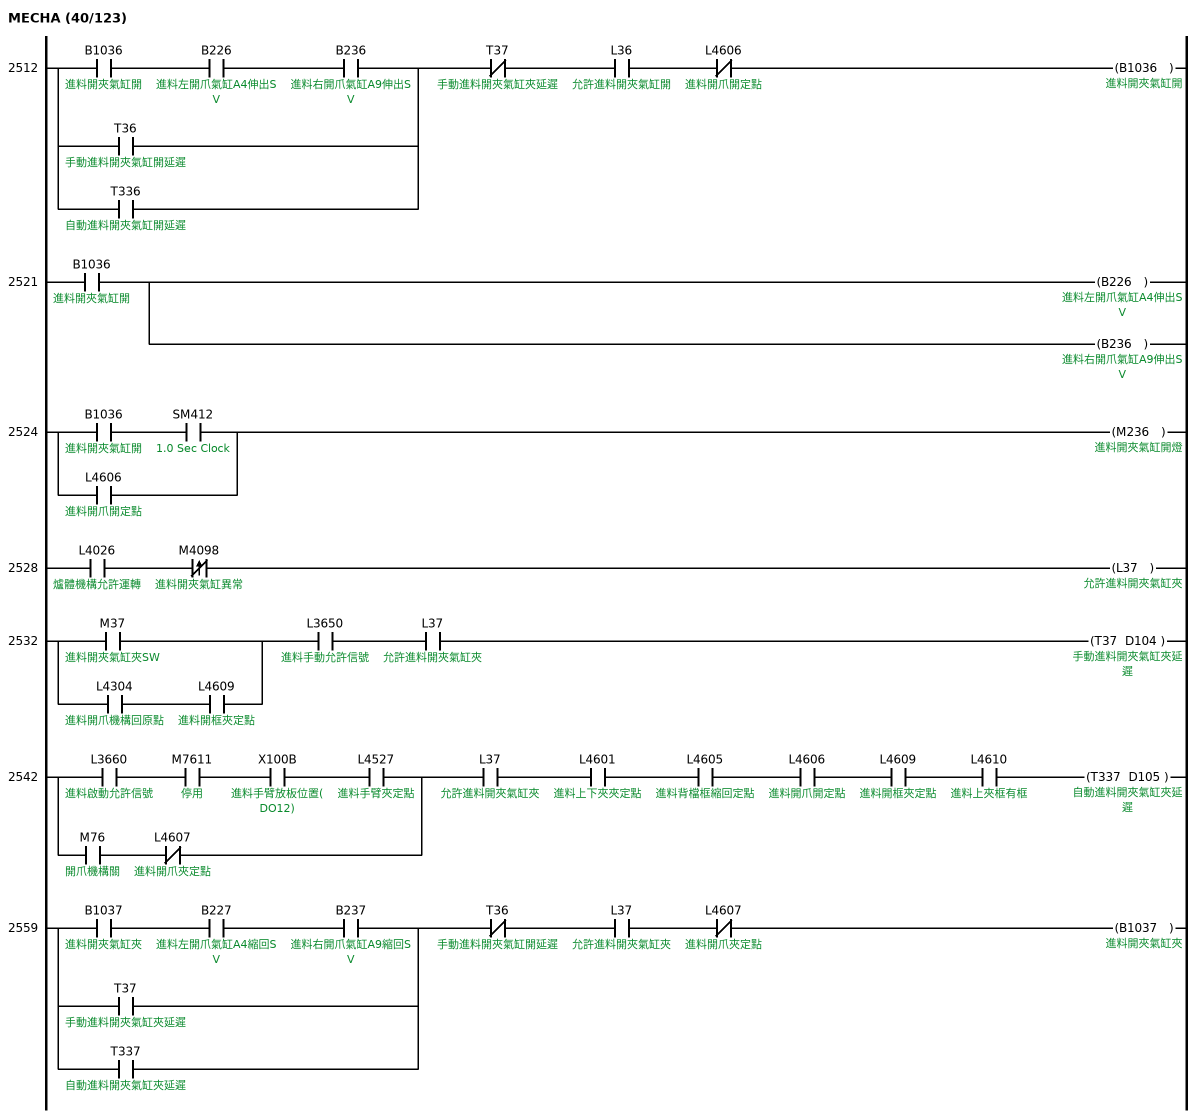
[picture p336: ladder of MECHA, rungs at steps 2512 to 2559]
2512  LD      B1036  ; 進料開夾氣缸開
      AND     B226  ; 進料左開爪氣缸A4伸出SV
      AND     B236  ; 進料右開爪氣缸A9伸出SV
      OR      T36  ; 手動進料開夾氣缸開延遲
      OR      T336  ; 自動進料開夾氣缸開延遲
      ANI     T37  ; 手動進料開夾氣缸夾延遲
      AND     L36  ; 允許進料開夾氣缸開
      ANI     L4606  ; 進料開爪開定點
      OUT     B1036  ; 進料開夾氣缸開
2521  LD      B1036  ; 進料開夾氣缸開
      OUT     B226  ; 進料左開爪氣缸A4伸出SV
      OUT     B236  ; 進料右開爪氣缸A9伸出SV
2524  LD      B1036  ; 進料開夾氣缸開
      AND     SM412  ; 1.0 Sec Clock
      OR      L4606  ; 進料開爪開定點
      OUT     M236  ; 進料開夾氣缸開燈
2528  LD      L4026  ; 爐體機構允許運轉
      ANDPI   M4098  ; 進料開夾氣缸異常
      OUT     L37  ; 允許進料開夾氣缸夾
2532  LD      M37  ; 進料開夾氣缸夾SW
      LD      L4304  ; 進料開爪機構回原點
      AND     L4609  ; 進料開框夾定點
      ORB
      AND     L3650  ; 進料手動允許信號
      AND     L37  ; 允許進料開夾氣缸夾
      OUT     T37 D104  ; 手動進料開夾氣缸夾延遲
2542  LD      L3660  ; 進料啟動允許信號
      AND     M7611  ; 停用
      AND     X100B  ; 進料手臂放板位置(DO12)
      AND     L4527  ; 進料手臂夾定點
      LD      M76  ; 開爪機構關
      ANI     L4607  ; 進料開爪夾定點
      ORB
      AND     L37  ; 允許進料開夾氣缸夾
      AND     L4601  ; 進料上下夾夾定點
      AND     L4605  ; 進料背檔框縮回定點
      AND     L4606  ; 進料開爪開定點
      AND     L4609  ; 進料開框夾定點
      AND     L4610  ; 進料上夾框有框
      OUT     T337 D105  ; 自動進料開夾氣缸夾延遲
2559  LD      B1037  ; 進料開夾氣缸夾
      AND     B227  ; 進料左開爪氣缸A4縮回SV
      AND     B237  ; 進料右開爪氣缸A9縮回SV
      OR      T37  ; 手動進料開夾氣缸夾延遲
      OR      T337  ; 自動進料開夾氣缸夾延遲
      ANI     T36  ; 手動進料開夾氣缸開延遲
      AND     L37  ; 允許進料開夾氣缸夾
      ANI     L4607  ; 進料開爪夾定點
      OUT     B1037  ; 進料開夾氣缸夾
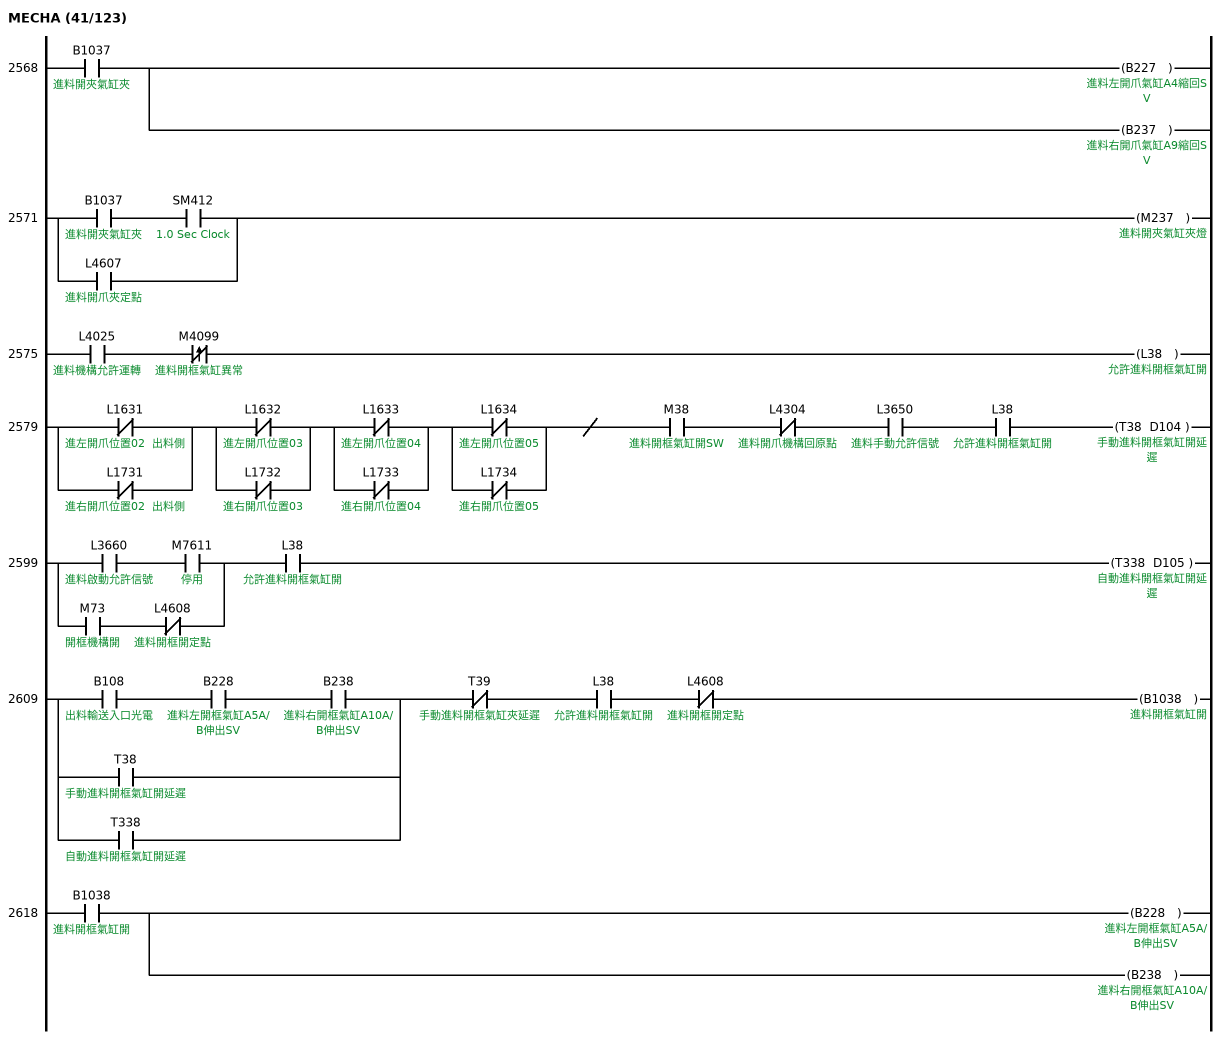
2568  LD      B1037  ; 進料開夾氣缸夾
      OUT     B227  ; 進料左開爪氣缸A4縮回SV
      OUT     B237  ; 進料右開爪氣缸A9縮回SV
2571  LD      B1037  ; 進料開夾氣缸夾
      AND     SM412  ; 1.0 Sec Clock
      OR      L4607  ; 進料開爪夾定點
      OUT     M237  ; 進料開夾氣缸夾燈
2575  LD      L4025  ; 進料機構允許運轉
      ANDPI   M4099  ; 進料開框氣缸異常
      OUT     L38  ; 允許進料開框氣缸開
2579  LDI     L1631  ; 進左開爪位置02  出料側
      ORI     L1731  ; 進右開爪位置02  出料側
      LDI     L1632  ; 進左開爪位置03
      ORI     L1732  ; 進右開爪位置03
      ANB
      LDI     L1633  ; 進左開爪位置04
      ORI     L1733  ; 進右開爪位置04
      ANB
      LDI     L1634  ; 進左開爪位置05
      ORI     L1734  ; 進右開爪位置05
      ANB
      INV
      AND     M38  ; 進料開框氣缸開SW
      ANI     L4304  ; 進料開爪機構回原點
      AND     L3650  ; 進料手動允許信號
      AND     L38  ; 允許進料開框氣缸開
      OUT     T38 D104  ; 手動進料開框氣缸開延遲
2599  LD      L3660  ; 進料啟動允許信號
      AND     M7611  ; 停用
      LD      M73  ; 開框機構開
      ANI     L4608  ; 進料開框開定點
      ORB
      AND     L38  ; 允許進料開框氣缸開
      OUT     T338 D105  ; 自動進料開框氣缸開延遲
2609  LD      B108  ; 出料輸送入口光電
      AND     B228  ; 進料左開框氣缸A5A/B伸出SV
      AND     B238  ; 進料右開框氣缸A10A/B伸出SV
      OR      T38  ; 手動進料開框氣缸開延遲
      OR      T338  ; 自動進料開框氣缸開延遲
      ANI     T39  ; 手動進料開框氣缸夾延遲
      AND     L38  ; 允許進料開框氣缸開
      ANI     L4608  ; 進料開框開定點
      OUT     B1038  ; 進料開框氣缸開
2618  LD      B1038  ; 進料開框氣缸開
      OUT     B228  ; 進料左開框氣缸A5A/B伸出SV
      OUT     B238  ; 進料右開框氣缸A10A/B伸出SV
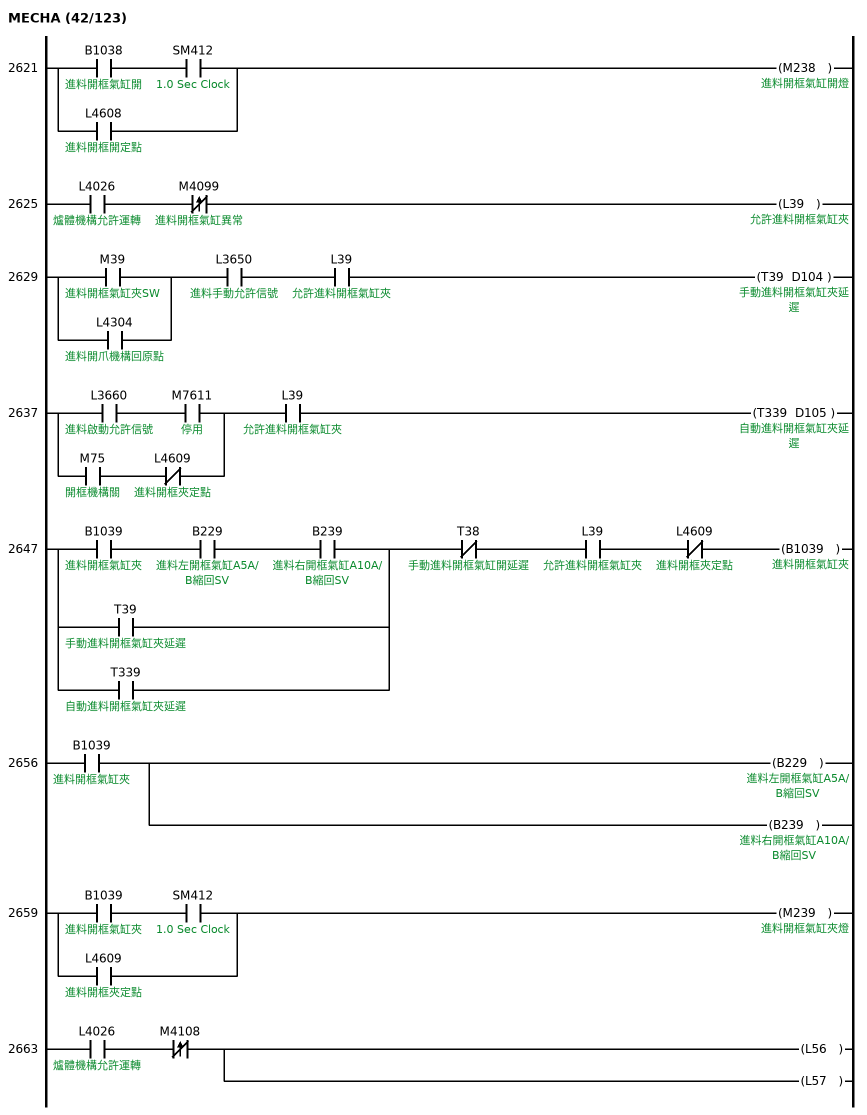
2621  LD      B1038  ; 進料開框氣缸開
      AND     SM412  ; 1.0 Sec Clock
      OR      L4608  ; 進料開框開定點
      OUT     M238  ; 進料開框氣缸開燈
2625  LD      L4026  ; 爐體機構允許運轉
      ANDPI   M4099  ; 進料開框氣缸異常
      OUT     L39  ; 允許進料開框氣缸夾
2629  LD      M39  ; 進料開框氣缸夾SW
      OR      L4304  ; 進料開爪機構回原點
      AND     L3650  ; 進料手動允許信號
      AND     L39  ; 允許進料開框氣缸夾
      OUT     T39 D104  ; 手動進料開框氣缸夾延遲
2637  LD      L3660  ; 進料啟動允許信號
      AND     M7611  ; 停用
      LD      M75  ; 開框機構關
      ANI     L4609  ; 進料開框夾定點
      ORB
      AND     L39  ; 允許進料開框氣缸夾
      OUT     T339 D105  ; 自動進料開框氣缸夾延遲
2647  LD      B1039  ; 進料開框氣缸夾
      AND     B229  ; 進料左開框氣缸A5A/B縮回SV
      AND     B239  ; 進料右開框氣缸A10A/B縮回SV
      OR      T39  ; 手動進料開框氣缸夾延遲
      OR      T339  ; 自動進料開框氣缸夾延遲
      ANI     T38  ; 手動進料開框氣缸開延遲
      AND     L39  ; 允許進料開框氣缸夾
      ANI     L4609  ; 進料開框夾定點
      OUT     B1039  ; 進料開框氣缸夾
2656  LD      B1039  ; 進料開框氣缸夾
      OUT     B229  ; 進料左開框氣缸A5A/B縮回SV
      OUT     B239  ; 進料右開框氣缸A10A/B縮回SV
2659  LD      B1039  ; 進料開框氣缸夾
      AND     SM412  ; 1.0 Sec Clock
      OR      L4609  ; 進料開框夾定點
      OUT     M239  ; 進料開框氣缸夾燈
2663  LD      L4026  ; 爐體機構允許運轉
      ANDPI   M4108
      OUT     L56
      OUT     L57
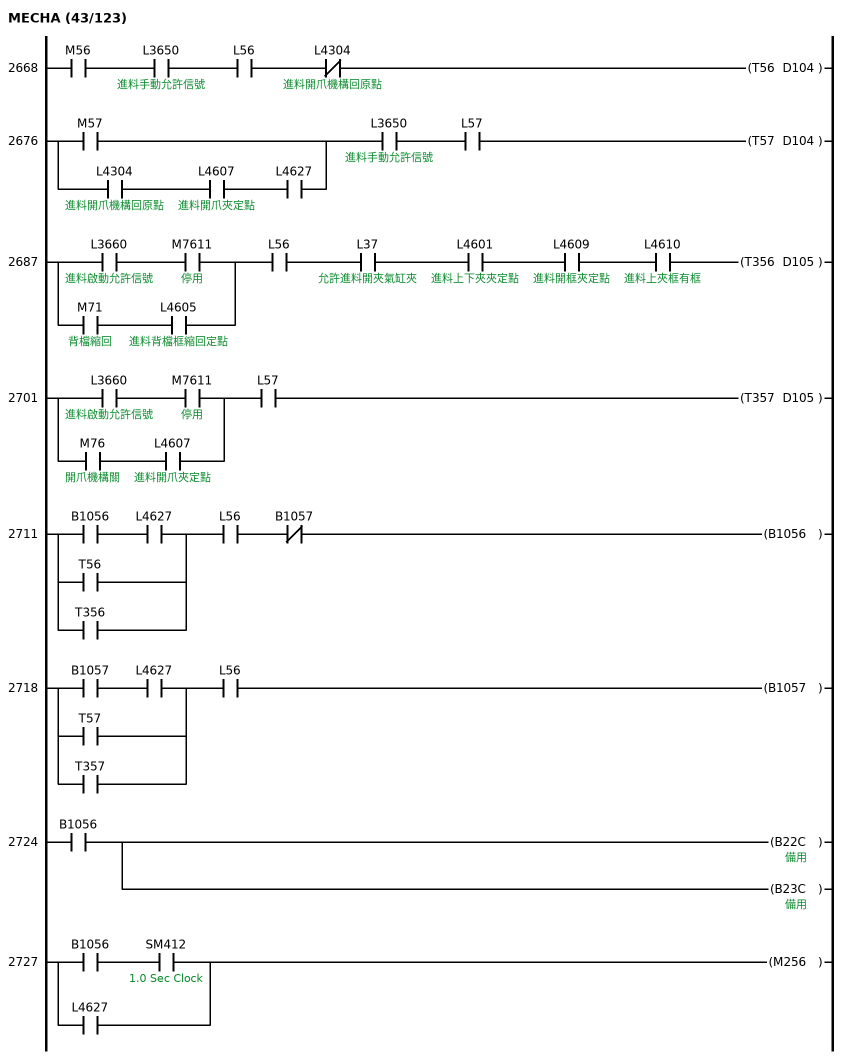
2668  LD      M56
      AND     L3650  ; 進料手動允許信號
      AND     L56
      ANI     L4304  ; 進料開爪機構回原點
      OUT     T56 D104
2676  LD      M57
      LD      L4304  ; 進料開爪機構回原點
      AND     L4607  ; 進料開爪夾定點
      AND     L4627
      ORB
      AND     L3650  ; 進料手動允許信號
      AND     L57
      OUT     T57 D104
2687  LD      L3660  ; 進料啟動允許信號
      AND     M7611  ; 停用
      LD      M71  ; 背檔縮回
      AND     L4605  ; 進料背檔框縮回定點
      ORB
      AND     L56
      AND     L37  ; 允許進料開夾氣缸夾
      AND     L4601  ; 進料上下夾夾定點
      AND     L4609  ; 進料開框夾定點
      AND     L4610  ; 進料上夾框有框
      OUT     T356 D105
2701  LD      L3660  ; 進料啟動允許信號
      AND     M7611  ; 停用
      LD      M76  ; 開爪機構關
      AND     L4607  ; 進料開爪夾定點
      ORB
      AND     L57
      OUT     T357 D105
2711  LD      B1056
      AND     L4627
      OR      T56
      OR      T356
      AND     L56
      ANI     B1057
      OUT     B1056
2718  LD      B1057
      AND     L4627
      OR      T57
      OR      T357
      AND     L56
      OUT     B1057
2724  LD      B1056
      OUT     B22C  ; 備用
      OUT     B23C  ; 備用
2727  LD      B1056
      AND     SM412  ; 1.0 Sec Clock
      OR      L4627
      OUT     M256
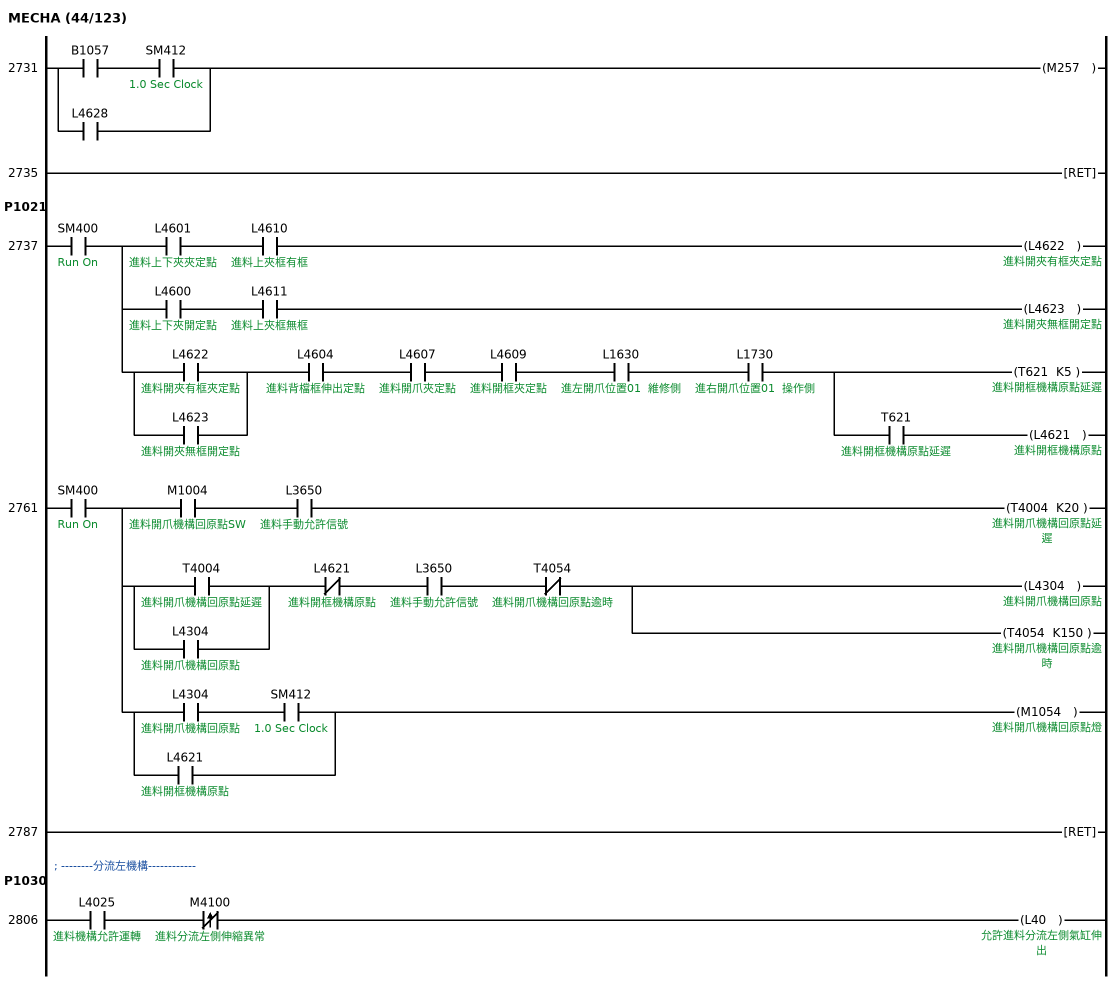
2731  LD      B1057
      AND     SM412  ; 1.0 Sec Clock
      OR      L4628
      OUT     M257
2735  RET
      P1021
2737  LD      SM400  ; Run On
      MPS
      AND     L4601  ; 進料上下夾夾定點
      AND     L4610  ; 進料上夾框有框
      OUT     L4622  ; 進料開夾有框夾定點
      MRD
      AND     L4600  ; 進料上下夾開定點
      AND     L4611  ; 進料上夾框無框
      OUT     L4623  ; 進料開夾無框開定點
      MPP
      LD      L4622  ; 進料開夾有框夾定點
      OR      L4623  ; 進料開夾無框開定點
      ANB
      AND     L4604  ; 進料背檔框伸出定點
      AND     L4607  ; 進料開爪夾定點
      AND     L4609  ; 進料開框夾定點
      AND     L1630  ; 進左開爪位置01  維修側
      AND     L1730  ; 進右開爪位置01  操作側
      OUT     T621 K5  ; 進料開框機構原點延遲
      AND     T621  ; 進料開框機構原點延遲
      OUT     L4621  ; 進料開框機構原點
2761  LD      SM400  ; Run On
      MPS
      AND     M1004  ; 進料開爪機構回原點SW
      AND     L3650  ; 進料手動允許信號
      OUT     T4004 K20  ; 進料開爪機構回原點延遲
      MRD
      LD      T4004  ; 進料開爪機構回原點延遲
      OR      L4304  ; 進料開爪機構回原點
      ANB
      ANI     L4621  ; 進料開框機構原點
      AND     L3650  ; 進料手動允許信號
      ANI     T4054  ; 進料開爪機構回原點逾時
      OUT     L4304  ; 進料開爪機構回原點
      OUT     T4054 K150  ; 進料開爪機構回原點逾時
      MPP
      LD      L4304  ; 進料開爪機構回原點
      AND     SM412  ; 1.0 Sec Clock
      OR      L4621  ; 進料開框機構原點
      ANB
      OUT     M1054  ; 進料開爪機構回原點燈
2787  RET
; --------分流左機構------------
      P1030
2806  LD      L4025  ; 進料機構允許運轉
      ANDPI   M4100  ; 進料分流左側伸縮異常
      OUT     L40  ; 允許進料分流左側氣缸伸出
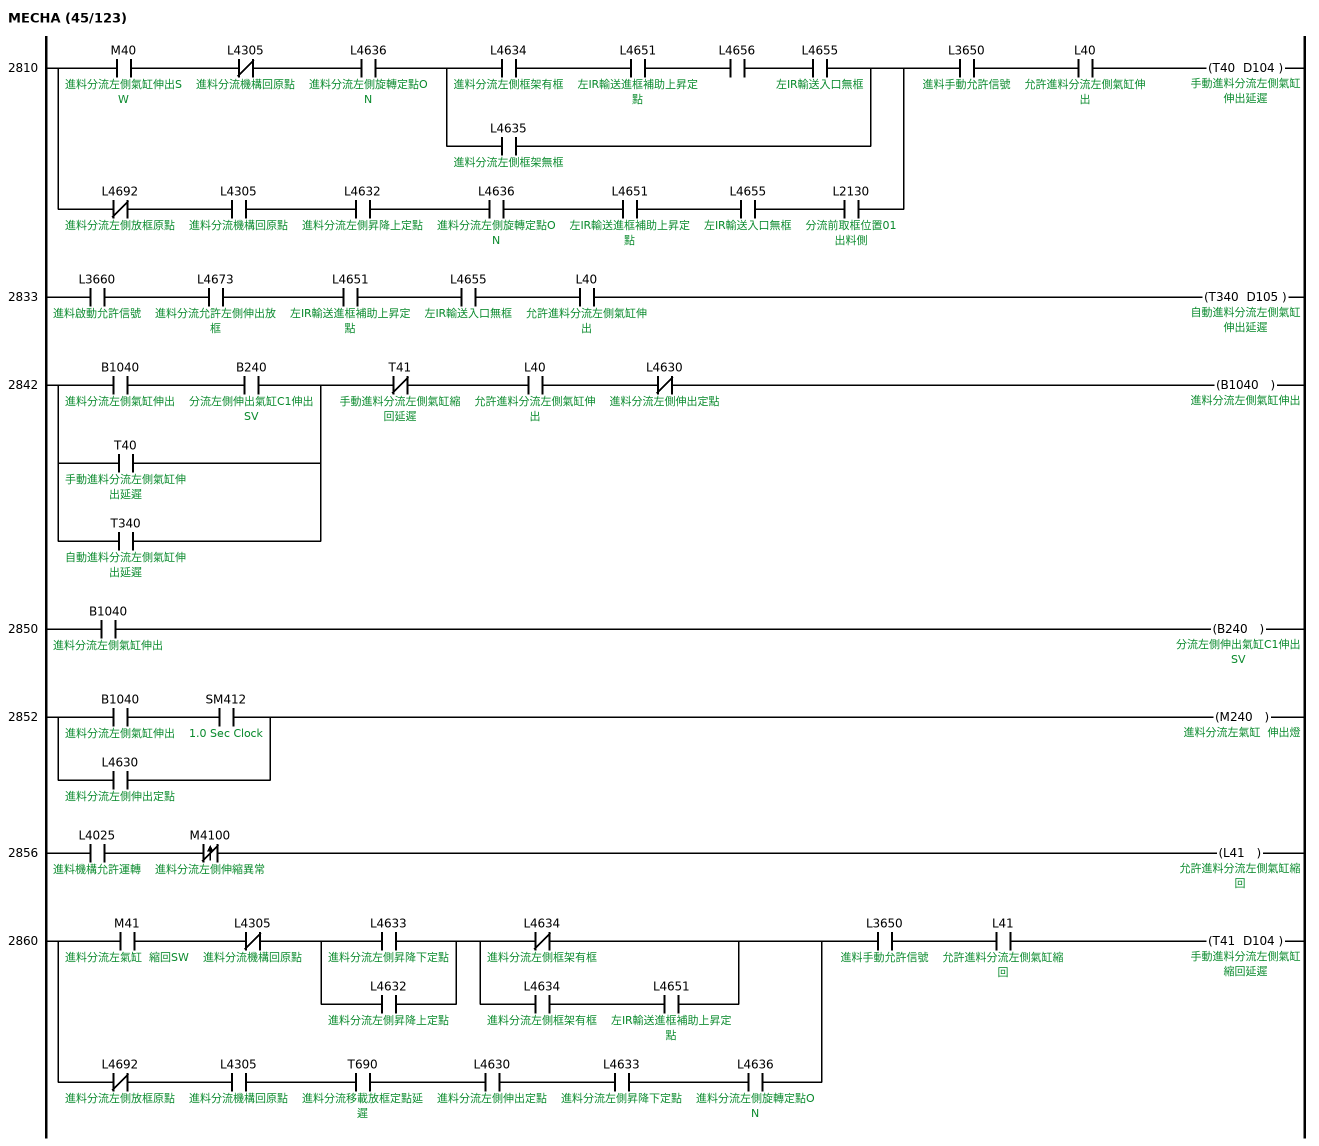
2810  LD      M40  ; 進料分流左側氣缸伸出SW
      ANI     L4305  ; 進料分流機構回原點
      AND     L4636  ; 進料分流左側旋轉定點ON
      LD      L4634  ; 進料分流左側框架有框
      AND     L4651  ; 左IR輸送進框補助上昇定點
      AND     L4656
      AND     L4655  ; 左IR輸送入口無框
      OR      L4635  ; 進料分流左側框架無框
      ANB
      LDI     L4692  ; 進料分流左側放框原點
      AND     L4305  ; 進料分流機構回原點
      AND     L4632  ; 進料分流左側昇降上定點
      AND     L4636  ; 進料分流左側旋轉定點ON
      AND     L4651  ; 左IR輸送進框補助上昇定點
      AND     L4655  ; 左IR輸送入口無框
      AND     L2130  ; 分流前取框位置01  出料側
      ORB
      AND     L3650  ; 進料手動允許信號
      AND     L40  ; 允許進料分流左側氣缸伸出
      OUT     T40 D104  ; 手動進料分流左側氣缸伸出延遲
2833  LD      L3660  ; 進料啟動允許信號
      AND     L4673  ; 進料分流允許左側伸出放框
      AND     L4651  ; 左IR輸送進框補助上昇定點
      AND     L4655  ; 左IR輸送入口無框
      AND     L40  ; 允許進料分流左側氣缸伸出
      OUT     T340 D105  ; 自動進料分流左側氣缸伸出延遲
2842  LD      B1040  ; 進料分流左側氣缸伸出
      AND     B240  ; 分流左側伸出氣缸C1伸出SV
      OR      T40  ; 手動進料分流左側氣缸伸出延遲
      OR      T340  ; 自動進料分流左側氣缸伸出延遲
      ANI     T41  ; 手動進料分流左側氣缸縮回延遲
      AND     L40  ; 允許進料分流左側氣缸伸出
      ANI     L4630  ; 進料分流左側伸出定點
      OUT     B1040  ; 進料分流左側氣缸伸出
2850  LD      B1040  ; 進料分流左側氣缸伸出
      OUT     B240  ; 分流左側伸出氣缸C1伸出SV
2852  LD      B1040  ; 進料分流左側氣缸伸出
      AND     SM412  ; 1.0 Sec Clock
      OR      L4630  ; 進料分流左側伸出定點
      OUT     M240  ; 進料分流左氣缸  伸出燈
2856  LD      L4025  ; 進料機構允許運轉
      ANDPI   M4100  ; 進料分流左側伸縮異常
      OUT     L41  ; 允許進料分流左側氣缸縮回
2860  LD      M41  ; 進料分流左氣缸  縮回SW
      ANI     L4305  ; 進料分流機構回原點
      LD      L4633  ; 進料分流左側昇降下定點
      OR      L4632  ; 進料分流左側昇降上定點
      ANB
      LDI     L4634  ; 進料分流左側框架有框
      LD      L4634  ; 進料分流左側框架有框
      AND     L4651  ; 左IR輸送進框補助上昇定點
      ORB
      ANB
      LDI     L4692  ; 進料分流左側放框原點
      AND     L4305  ; 進料分流機構回原點
      AND     T690  ; 進料分流移載放框定點延遲
      AND     L4630  ; 進料分流左側伸出定點
      AND     L4633  ; 進料分流左側昇降下定點
      AND     L4636  ; 進料分流左側旋轉定點ON
      ORB
      AND     L3650  ; 進料手動允許信號
      AND     L41  ; 允許進料分流左側氣缸縮回
      OUT     T41 D104  ; 手動進料分流左側氣缸縮回延遲
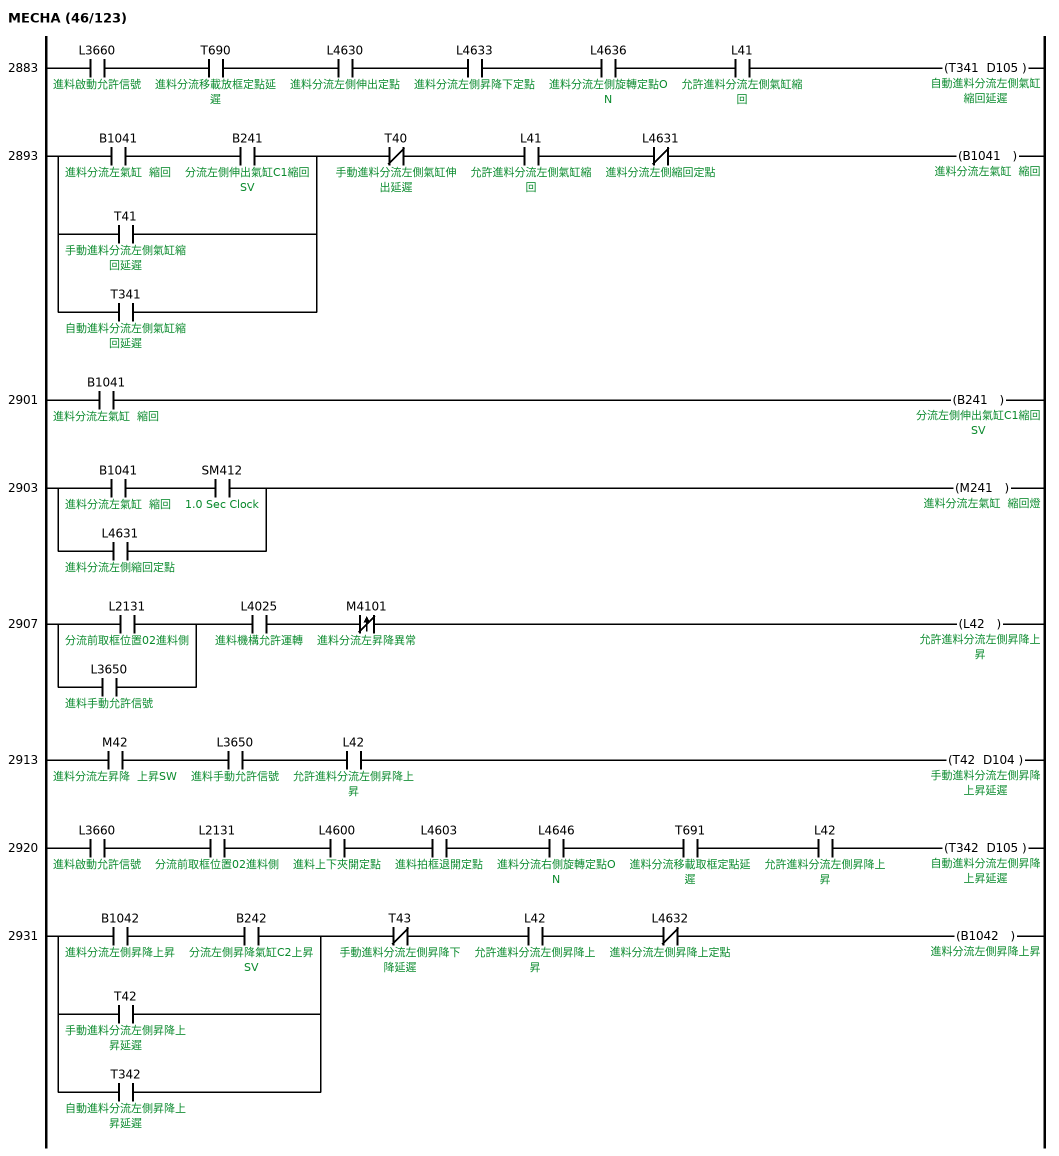
2883  LD      L3660  ; 進料啟動允許信號
      AND     T690  ; 進料分流移載放框定點延遲
      AND     L4630  ; 進料分流左側伸出定點
      AND     L4633  ; 進料分流左側昇降下定點
      AND     L4636  ; 進料分流左側旋轉定點ON
      AND     L41  ; 允許進料分流左側氣缸縮回
      OUT     T341 D105  ; 自動進料分流左側氣缸縮回延遲
2893  LD      B1041  ; 進料分流左氣缸  縮回
      AND     B241  ; 分流左側伸出氣缸C1縮回SV
      OR      T41  ; 手動進料分流左側氣缸縮回延遲
      OR      T341  ; 自動進料分流左側氣缸縮回延遲
      ANI     T40  ; 手動進料分流左側氣缸伸出延遲
      AND     L41  ; 允許進料分流左側氣缸縮回
      ANI     L4631  ; 進料分流左側縮回定點
      OUT     B1041  ; 進料分流左氣缸  縮回
2901  LD      B1041  ; 進料分流左氣缸  縮回
      OUT     B241  ; 分流左側伸出氣缸C1縮回SV
2903  LD      B1041  ; 進料分流左氣缸  縮回
      AND     SM412  ; 1.0 Sec Clock
      OR      L4631  ; 進料分流左側縮回定點
      OUT     M241  ; 進料分流左氣缸  縮回燈
2907  LD      L2131  ; 分流前取框位置02進料側
      OR      L3650  ; 進料手動允許信號
      AND     L4025  ; 進料機構允許運轉
      ANDPI   M4101  ; 進料分流左昇降異常
      OUT     L42  ; 允許進料分流左側昇降上昇
2913  LD      M42  ; 進料分流左昇降  上昇SW
      AND     L3650  ; 進料手動允許信號
      AND     L42  ; 允許進料分流左側昇降上昇
      OUT     T42 D104  ; 手動進料分流左側昇降上昇延遲
2920  LD      L3660  ; 進料啟動允許信號
      AND     L2131  ; 分流前取框位置02進料側
      AND     L4600  ; 進料上下夾開定點
      AND     L4603  ; 進料拍框退開定點
      AND     L4646  ; 進料分流右側旋轉定點ON
      AND     T691  ; 進料分流移載取框定點延遲
      AND     L42  ; 允許進料分流左側昇降上昇
      OUT     T342 D105  ; 自動進料分流左側昇降上昇延遲
2931  LD      B1042  ; 進料分流左側昇降上昇
      AND     B242  ; 分流左側昇降氣缸C2上昇SV
      OR      T42  ; 手動進料分流左側昇降上昇延遲
      OR      T342  ; 自動進料分流左側昇降上昇延遲
      ANI     T43  ; 手動進料分流左側昇降下降延遲
      AND     L42  ; 允許進料分流左側昇降上昇
      ANI     L4632  ; 進料分流左側昇降上定點
      OUT     B1042  ; 進料分流左側昇降上昇
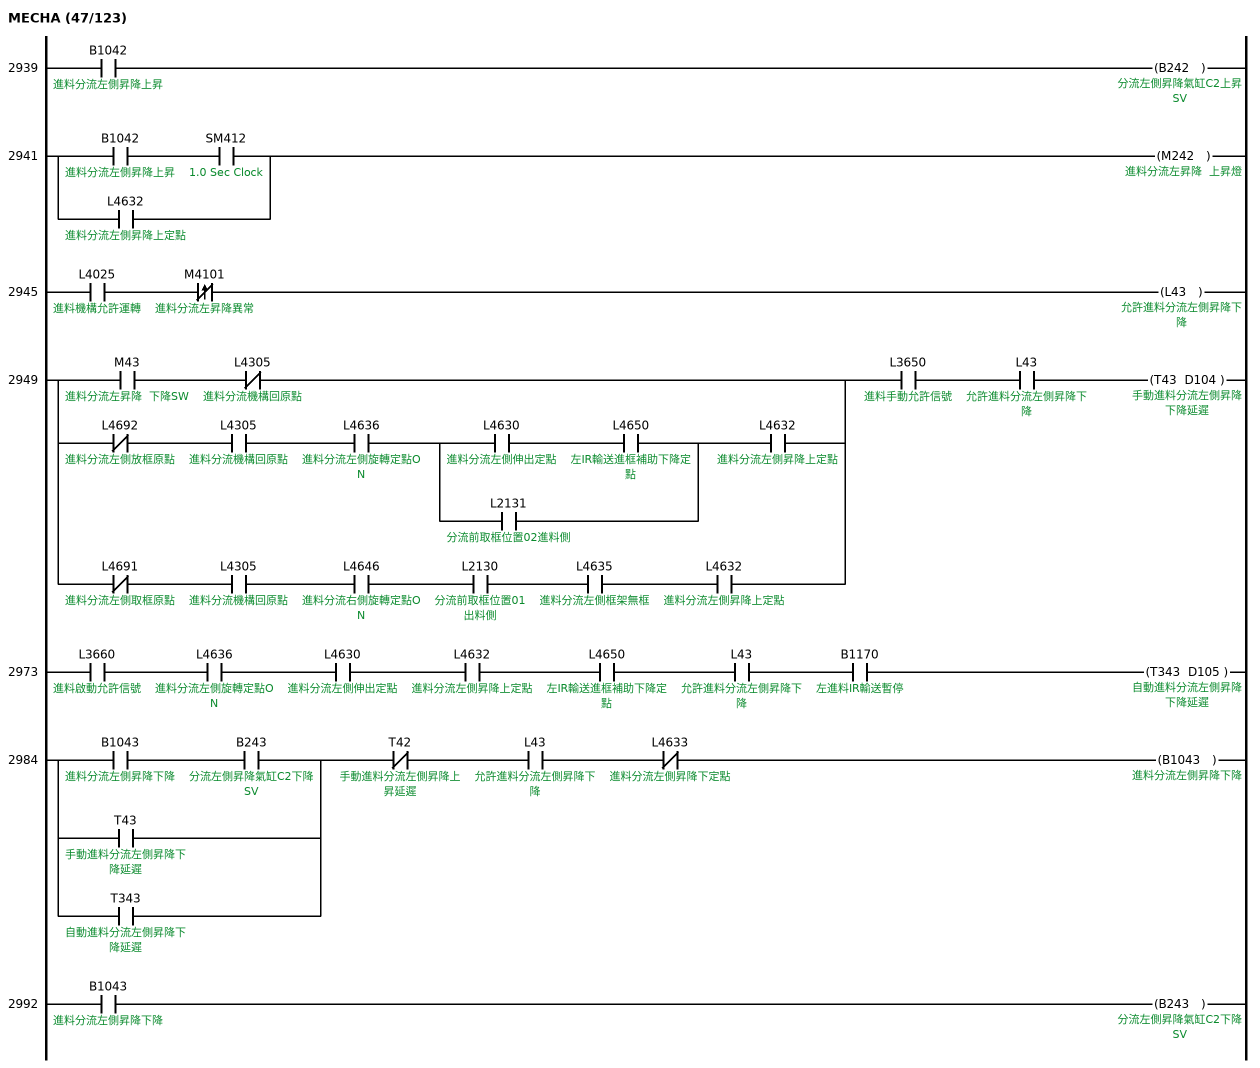
2939  LD      B1042  ; 進料分流左側昇降上昇
      OUT     B242  ; 分流左側昇降氣缸C2上昇SV
2941  LD      B1042  ; 進料分流左側昇降上昇
      AND     SM412  ; 1.0 Sec Clock
      OR      L4632  ; 進料分流左側昇降上定點
      OUT     M242  ; 進料分流左昇降  上昇燈
2945  LD      L4025  ; 進料機構允許運轉
      ANDPI   M4101  ; 進料分流左昇降異常
      OUT     L43  ; 允許進料分流左側昇降下降
2949  LD      M43  ; 進料分流左昇降  下降SW
      ANI     L4305  ; 進料分流機構回原點
      LDI     L4692  ; 進料分流左側放框原點
      AND     L4305  ; 進料分流機構回原點
      AND     L4636  ; 進料分流左側旋轉定點ON
      LD      L4630  ; 進料分流左側伸出定點
      AND     L4650  ; 左IR輸送進框補助下降定點
      OR      L2131  ; 分流前取框位置02進料側
      ANB
      AND     L4632  ; 進料分流左側昇降上定點
      ORB
      LDI     L4691  ; 進料分流左側取框原點
      AND     L4305  ; 進料分流機構回原點
      AND     L4646  ; 進料分流右側旋轉定點ON
      AND     L2130  ; 分流前取框位置01  出料側
      AND     L4635  ; 進料分流左側框架無框
      AND     L4632  ; 進料分流左側昇降上定點
      ORB
      AND     L3650  ; 進料手動允許信號
      AND     L43  ; 允許進料分流左側昇降下降
      OUT     T43 D104  ; 手動進料分流左側昇降下降延遲
2973  LD      L3660  ; 進料啟動允許信號
      AND     L4636  ; 進料分流左側旋轉定點ON
      AND     L4630  ; 進料分流左側伸出定點
      AND     L4632  ; 進料分流左側昇降上定點
      AND     L4650  ; 左IR輸送進框補助下降定點
      AND     L43  ; 允許進料分流左側昇降下降
      AND     B1170  ; 左進料IR輸送暫停
      OUT     T343 D105  ; 自動進料分流左側昇降下降延遲
2984  LD      B1043  ; 進料分流左側昇降下降
      AND     B243  ; 分流左側昇降氣缸C2下降SV
      OR      T43  ; 手動進料分流左側昇降下降延遲
      OR      T343  ; 自動進料分流左側昇降下降延遲
      ANI     T42  ; 手動進料分流左側昇降上昇延遲
      AND     L43  ; 允許進料分流左側昇降下降
      ANI     L4633  ; 進料分流左側昇降下定點
      OUT     B1043  ; 進料分流左側昇降下降
2992  LD      B1043  ; 進料分流左側昇降下降
      OUT     B243  ; 分流左側昇降氣缸C2下降SV
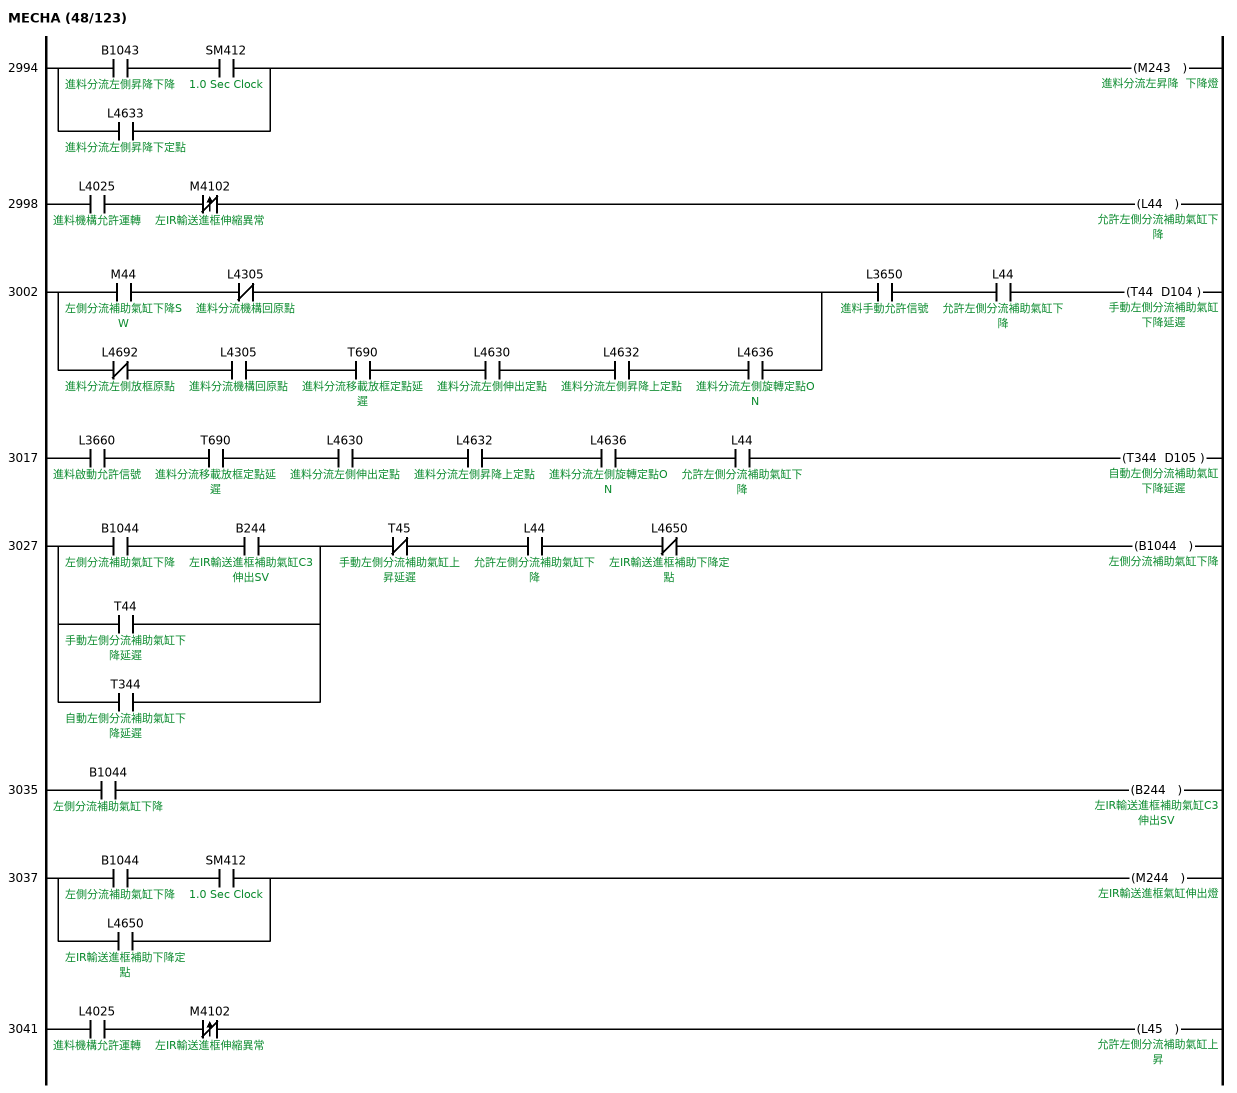
2994  LD      B1043  ; 進料分流左側昇降下降
      AND     SM412  ; 1.0 Sec Clock
      OR      L4633  ; 進料分流左側昇降下定點
      OUT     M243  ; 進料分流左昇降  下降燈
2998  LD      L4025  ; 進料機構允許運轉
      ANDPI   M4102  ; 左IR輸送進框伸縮異常
      OUT     L44  ; 允許左側分流補助氣缸下降
3002  LD      M44  ; 左側分流補助氣缸下降SW
      ANI     L4305  ; 進料分流機構回原點
      LDI     L4692  ; 進料分流左側放框原點
      AND     L4305  ; 進料分流機構回原點
      AND     T690  ; 進料分流移載放框定點延遲
      AND     L4630  ; 進料分流左側伸出定點
      AND     L4632  ; 進料分流左側昇降上定點
      AND     L4636  ; 進料分流左側旋轉定點ON
      ORB
      AND     L3650  ; 進料手動允許信號
      AND     L44  ; 允許左側分流補助氣缸下降
      OUT     T44 D104  ; 手動左側分流補助氣缸下降延遲
3017  LD      L3660  ; 進料啟動允許信號
      AND     T690  ; 進料分流移載放框定點延遲
      AND     L4630  ; 進料分流左側伸出定點
      AND     L4632  ; 進料分流左側昇降上定點
      AND     L4636  ; 進料分流左側旋轉定點ON
      AND     L44  ; 允許左側分流補助氣缸下降
      OUT     T344 D105  ; 自動左側分流補助氣缸下降延遲
3027  LD      B1044  ; 左側分流補助氣缸下降
      AND     B244  ; 左IR輸送進框補助氣缸C3伸出SV
      OR      T44  ; 手動左側分流補助氣缸下降延遲
      OR      T344  ; 自動左側分流補助氣缸下降延遲
      ANI     T45  ; 手動左側分流補助氣缸上昇延遲
      AND     L44  ; 允許左側分流補助氣缸下降
      ANI     L4650  ; 左IR輸送進框補助下降定點
      OUT     B1044  ; 左側分流補助氣缸下降
3035  LD      B1044  ; 左側分流補助氣缸下降
      OUT     B244  ; 左IR輸送進框補助氣缸C3伸出SV
3037  LD      B1044  ; 左側分流補助氣缸下降
      AND     SM412  ; 1.0 Sec Clock
      OR      L4650  ; 左IR輸送進框補助下降定點
      OUT     M244  ; 左IR輸送進框氣缸伸出燈
3041  LD      L4025  ; 進料機構允許運轉
      ANDPI   M4102  ; 左IR輸送進框伸縮異常
      OUT     L45  ; 允許左側分流補助氣缸上昇
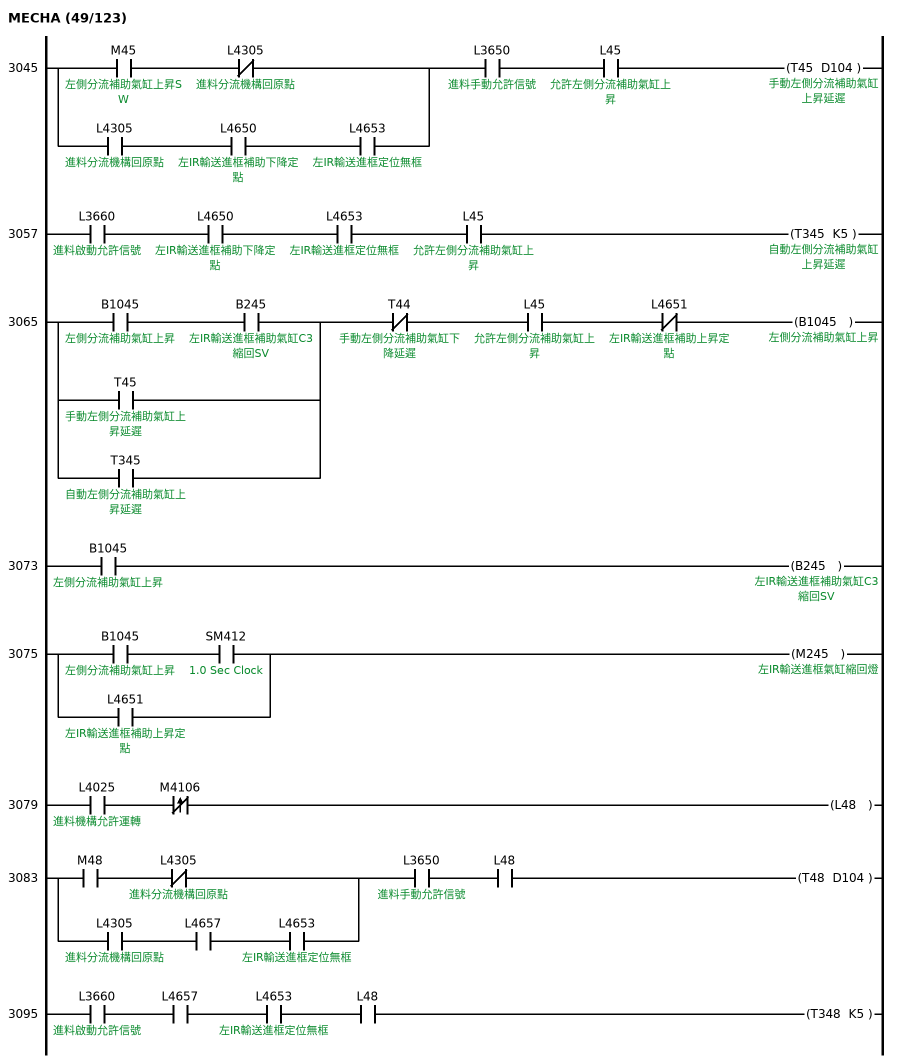
3045  LD      M45  ; 左側分流補助氣缸上昇SW
      ANI     L4305  ; 進料分流機構回原點
      LD      L4305  ; 進料分流機構回原點
      AND     L4650  ; 左IR輸送進框補助下降定點
      AND     L4653  ; 左IR輸送進框定位無框
      ORB
      AND     L3650  ; 進料手動允許信號
      AND     L45  ; 允許左側分流補助氣缸上昇
      OUT     T45 D104  ; 手動左側分流補助氣缸上昇延遲
3057  LD      L3660  ; 進料啟動允許信號
      AND     L4650  ; 左IR輸送進框補助下降定點
      AND     L4653  ; 左IR輸送進框定位無框
      AND     L45  ; 允許左側分流補助氣缸上昇
      OUT     T345 K5  ; 自動左側分流補助氣缸上昇延遲
3065  LD      B1045  ; 左側分流補助氣缸上昇
      AND     B245  ; 左IR輸送進框補助氣缸C3縮回SV
      OR      T45  ; 手動左側分流補助氣缸上昇延遲
      OR      T345  ; 自動左側分流補助氣缸上昇延遲
      ANI     T44  ; 手動左側分流補助氣缸下降延遲
      AND     L45  ; 允許左側分流補助氣缸上昇
      ANI     L4651  ; 左IR輸送進框補助上昇定點
      OUT     B1045  ; 左側分流補助氣缸上昇
3073  LD      B1045  ; 左側分流補助氣缸上昇
      OUT     B245  ; 左IR輸送進框補助氣缸C3縮回SV
3075  LD      B1045  ; 左側分流補助氣缸上昇
      AND     SM412  ; 1.0 Sec Clock
      OR      L4651  ; 左IR輸送進框補助上昇定點
      OUT     M245  ; 左IR輸送進框氣缸縮回燈
3079  LD      L4025  ; 進料機構允許運轉
      ANDPI   M4106
      OUT     L48
3083  LD      M48
      ANI     L4305  ; 進料分流機構回原點
      LD      L4305  ; 進料分流機構回原點
      AND     L4657
      AND     L4653  ; 左IR輸送進框定位無框
      ORB
      AND     L3650  ; 進料手動允許信號
      AND     L48
      OUT     T48 D104
3095  LD      L3660  ; 進料啟動允許信號
      AND     L4657
      AND     L4653  ; 左IR輸送進框定位無框
      AND     L48
      OUT     T348 K5
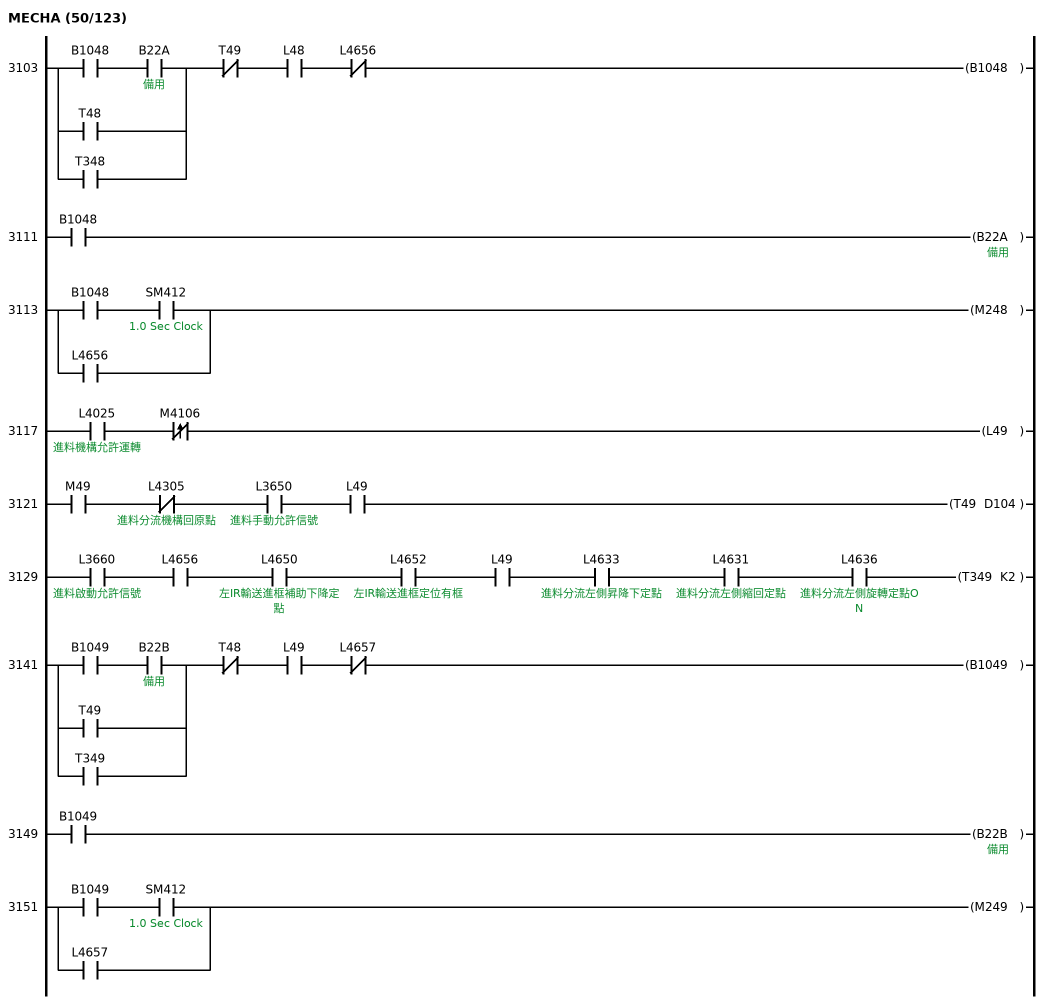
3103  LD      B1048
      AND     B22A  ; 備用
      OR      T48
      OR      T348
      ANI     T49
      AND     L48
      ANI     L4656
      OUT     B1048
3111  LD      B1048
      OUT     B22A  ; 備用
3113  LD      B1048
      AND     SM412  ; 1.0 Sec Clock
      OR      L4656
      OUT     M248
3117  LD      L4025  ; 進料機構允許運轉
      ANDPI   M4106
      OUT     L49
3121  LD      M49
      ANI     L4305  ; 進料分流機構回原點
      AND     L3650  ; 進料手動允許信號
      AND     L49
      OUT     T49 D104
3129  LD      L3660  ; 進料啟動允許信號
      AND     L4656
      AND     L4650  ; 左IR輸送進框補助下降定點
      AND     L4652  ; 左IR輸送進框定位有框
      AND     L49
      AND     L4633  ; 進料分流左側昇降下定點
      AND     L4631  ; 進料分流左側縮回定點
      AND     L4636  ; 進料分流左側旋轉定點ON
      OUT     T349 K2
3141  LD      B1049
      AND     B22B  ; 備用
      OR      T49
      OR      T349
      ANI     T48
      AND     L49
      ANI     L4657
      OUT     B1049
3149  LD      B1049
      OUT     B22B  ; 備用
3151  LD      B1049
      AND     SM412  ; 1.0 Sec Clock
      OR      L4657
      OUT     M249
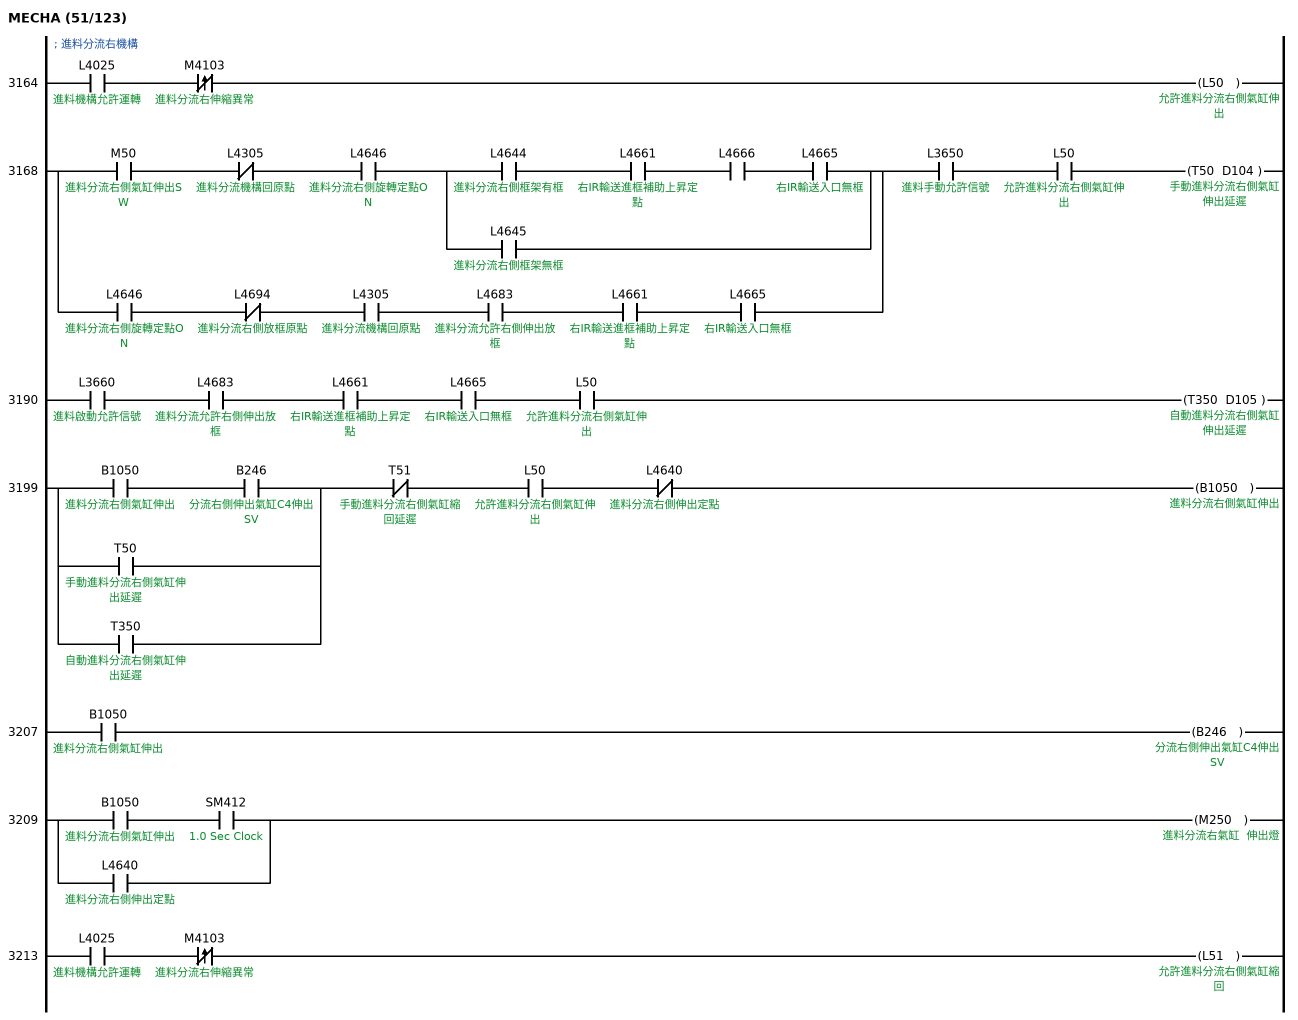
; 進料分流右機構
3164  LD      L4025  ; 進料機構允許運轉
      ANDPI   M4103  ; 進料分流右伸縮異常
      OUT     L50  ; 允許進料分流右側氣缸伸出
3168  LD      M50  ; 進料分流右側氣缸伸出SW
      ANI     L4305  ; 進料分流機構回原點
      AND     L4646  ; 進料分流右側旋轉定點ON
      LD      L4644  ; 進料分流右側框架有框
      AND     L4661  ; 右IR輸送進框補助上昇定點
      AND     L4666
      AND     L4665  ; 右IR輸送入口無框
      OR      L4645  ; 進料分流右側框架無框
      ANB
      LD      L4646  ; 進料分流右側旋轉定點ON
      ANI     L4694  ; 進料分流右側放框原點
      AND     L4305  ; 進料分流機構回原點
      AND     L4683  ; 進料分流允許右側伸出放框
      AND     L4661  ; 右IR輸送進框補助上昇定點
      AND     L4665  ; 右IR輸送入口無框
      ORB
      AND     L3650  ; 進料手動允許信號
      AND     L50  ; 允許進料分流右側氣缸伸出
      OUT     T50 D104  ; 手動進料分流右側氣缸伸出延遲
3190  LD      L3660  ; 進料啟動允許信號
      AND     L4683  ; 進料分流允許右側伸出放框
      AND     L4661  ; 右IR輸送進框補助上昇定點
      AND     L4665  ; 右IR輸送入口無框
      AND     L50  ; 允許進料分流右側氣缸伸出
      OUT     T350 D105  ; 自動進料分流右側氣缸伸出延遲
3199  LD      B1050  ; 進料分流右側氣缸伸出
      AND     B246  ; 分流右側伸出氣缸C4伸出SV
      OR      T50  ; 手動進料分流右側氣缸伸出延遲
      OR      T350  ; 自動進料分流右側氣缸伸出延遲
      ANI     T51  ; 手動進料分流右側氣缸縮回延遲
      AND     L50  ; 允許進料分流右側氣缸伸出
      ANI     L4640  ; 進料分流右側伸出定點
      OUT     B1050  ; 進料分流右側氣缸伸出
3207  LD      B1050  ; 進料分流右側氣缸伸出
      OUT     B246  ; 分流右側伸出氣缸C4伸出SV
3209  LD      B1050  ; 進料分流右側氣缸伸出
      AND     SM412  ; 1.0 Sec Clock
      OR      L4640  ; 進料分流右側伸出定點
      OUT     M250  ; 進料分流右氣缸  伸出燈
3213  LD      L4025  ; 進料機構允許運轉
      ANDPI   M4103  ; 進料分流右伸縮異常
      OUT     L51  ; 允許進料分流右側氣缸縮回
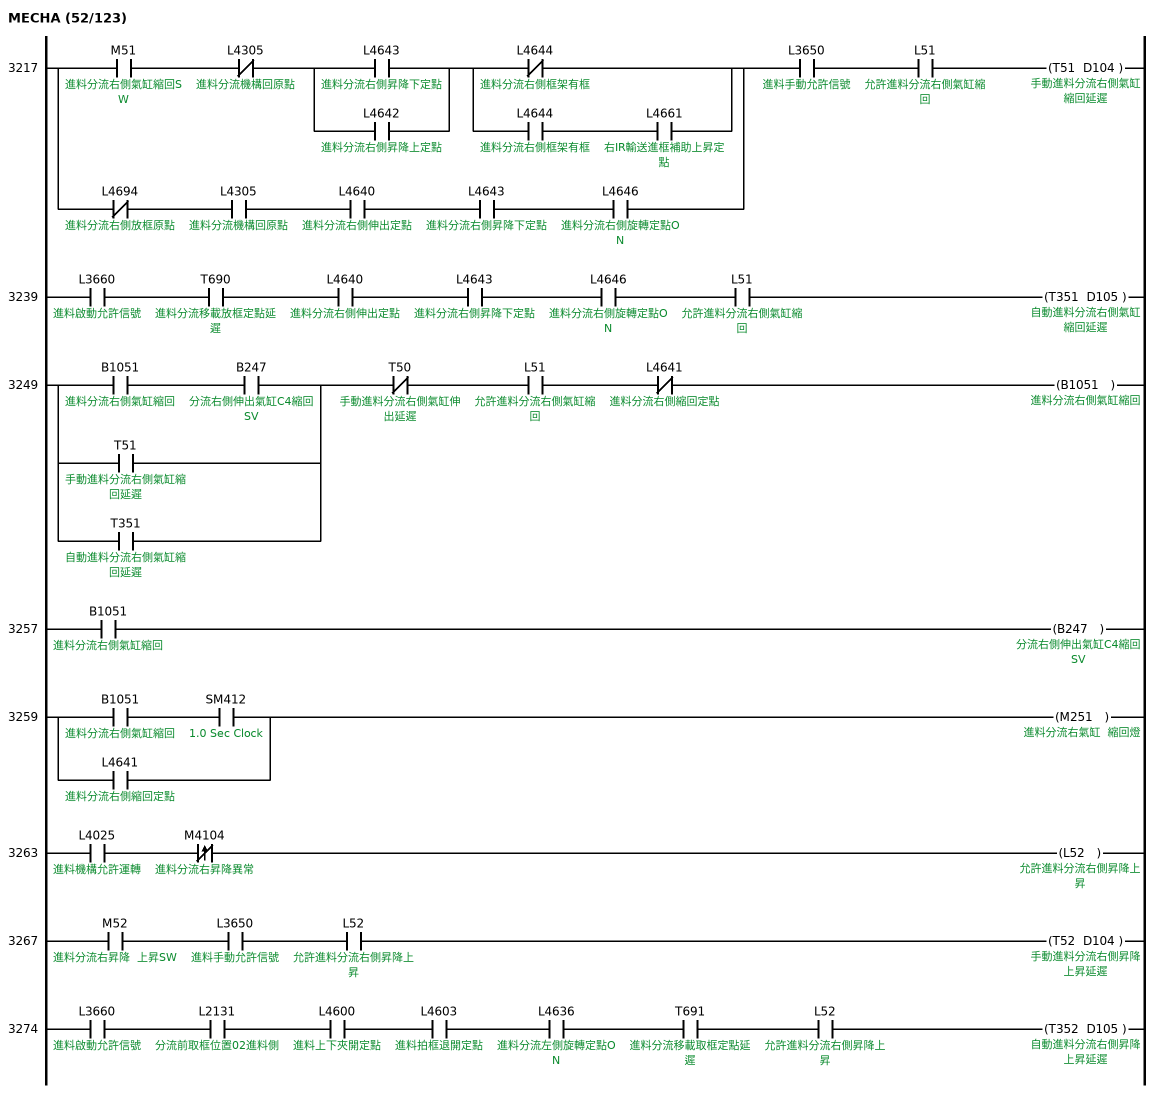
3217  LD      M51  ; 進料分流右側氣缸縮回SW
      ANI     L4305  ; 進料分流機構回原點
      LD      L4643  ; 進料分流右側昇降下定點
      OR      L4642  ; 進料分流右側昇降上定點
      ANB
      LDI     L4644  ; 進料分流右側框架有框
      LD      L4644  ; 進料分流右側框架有框
      AND     L4661  ; 右IR輸送進框補助上昇定點
      ORB
      ANB
      LDI     L4694  ; 進料分流右側放框原點
      AND     L4305  ; 進料分流機構回原點
      AND     L4640  ; 進料分流右側伸出定點
      AND     L4643  ; 進料分流右側昇降下定點
      AND     L4646  ; 進料分流右側旋轉定點ON
      ORB
      AND     L3650  ; 進料手動允許信號
      AND     L51  ; 允許進料分流右側氣缸縮回
      OUT     T51 D104  ; 手動進料分流右側氣缸縮回延遲
3239  LD      L3660  ; 進料啟動允許信號
      AND     T690  ; 進料分流移載放框定點延遲
      AND     L4640  ; 進料分流右側伸出定點
      AND     L4643  ; 進料分流右側昇降下定點
      AND     L4646  ; 進料分流右側旋轉定點ON
      AND     L51  ; 允許進料分流右側氣缸縮回
      OUT     T351 D105  ; 自動進料分流右側氣缸縮回延遲
3249  LD      B1051  ; 進料分流右側氣缸縮回
      AND     B247  ; 分流右側伸出氣缸C4縮回SV
      OR      T51  ; 手動進料分流右側氣缸縮回延遲
      OR      T351  ; 自動進料分流右側氣缸縮回延遲
      ANI     T50  ; 手動進料分流右側氣缸伸出延遲
      AND     L51  ; 允許進料分流右側氣缸縮回
      ANI     L4641  ; 進料分流右側縮回定點
      OUT     B1051  ; 進料分流右側氣缸縮回
3257  LD      B1051  ; 進料分流右側氣缸縮回
      OUT     B247  ; 分流右側伸出氣缸C4縮回SV
3259  LD      B1051  ; 進料分流右側氣缸縮回
      AND     SM412  ; 1.0 Sec Clock
      OR      L4641  ; 進料分流右側縮回定點
      OUT     M251  ; 進料分流右氣缸  縮回燈
3263  LD      L4025  ; 進料機構允許運轉
      ANDPI   M4104  ; 進料分流右昇降異常
      OUT     L52  ; 允許進料分流右側昇降上昇
3267  LD      M52  ; 進料分流右昇降  上昇SW
      AND     L3650  ; 進料手動允許信號
      AND     L52  ; 允許進料分流右側昇降上昇
      OUT     T52 D104  ; 手動進料分流右側昇降上昇延遲
3274  LD      L3660  ; 進料啟動允許信號
      AND     L2131  ; 分流前取框位置02進料側
      AND     L4600  ; 進料上下夾開定點
      AND     L4603  ; 進料拍框退開定點
      AND     L4636  ; 進料分流左側旋轉定點ON
      AND     T691  ; 進料分流移載取框定點延遲
      AND     L52  ; 允許進料分流右側昇降上昇
      OUT     T352 D105  ; 自動進料分流右側昇降上昇延遲
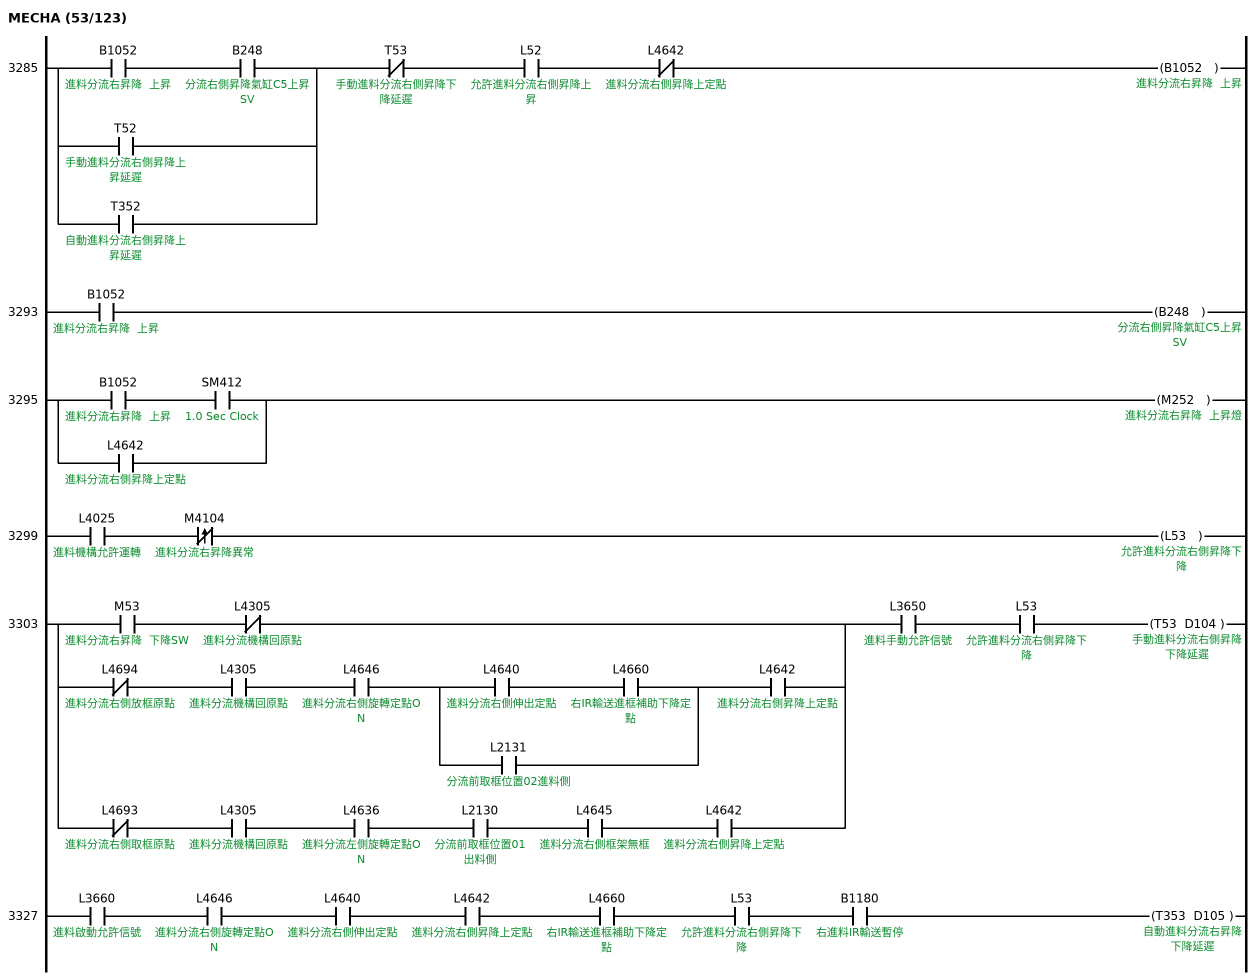
3285  LD      B1052  ; 進料分流右昇降  上昇
      AND     B248  ; 分流右側昇降氣缸C5上昇SV
      OR      T52  ; 手動進料分流右側昇降上昇延遲
      OR      T352  ; 自動進料分流右側昇降上昇延遲
      ANI     T53  ; 手動進料分流右側昇降下降延遲
      AND     L52  ; 允許進料分流右側昇降上昇
      ANI     L4642  ; 進料分流右側昇降上定點
      OUT     B1052  ; 進料分流右昇降  上昇
3293  LD      B1052  ; 進料分流右昇降  上昇
      OUT     B248  ; 分流右側昇降氣缸C5上昇SV
3295  LD      B1052  ; 進料分流右昇降  上昇
      AND     SM412  ; 1.0 Sec Clock
      OR      L4642  ; 進料分流右側昇降上定點
      OUT     M252  ; 進料分流右昇降  上昇燈
3299  LD      L4025  ; 進料機構允許運轉
      ANDPI   M4104  ; 進料分流右昇降異常
      OUT     L53  ; 允許進料分流右側昇降下降
3303  LD      M53  ; 進料分流右昇降  下降SW
      ANI     L4305  ; 進料分流機構回原點
      LDI     L4694  ; 進料分流右側放框原點
      AND     L4305  ; 進料分流機構回原點
      AND     L4646  ; 進料分流右側旋轉定點ON
      LD      L4640  ; 進料分流右側伸出定點
      AND     L4660  ; 右IR輸送進框補助下降定點
      OR      L2131  ; 分流前取框位置02進料側
      ANB
      AND     L4642  ; 進料分流右側昇降上定點
      ORB
      LDI     L4693  ; 進料分流右側取框原點
      AND     L4305  ; 進料分流機構回原點
      AND     L4636  ; 進料分流左側旋轉定點ON
      AND     L2130  ; 分流前取框位置01  出料側
      AND     L4645  ; 進料分流右側框架無框
      AND     L4642  ; 進料分流右側昇降上定點
      ORB
      AND     L3650  ; 進料手動允許信號
      AND     L53  ; 允許進料分流右側昇降下降
      OUT     T53 D104  ; 手動進料分流右側昇降下降延遲
3327  LD      L3660  ; 進料啟動允許信號
      AND     L4646  ; 進料分流右側旋轉定點ON
      AND     L4640  ; 進料分流右側伸出定點
      AND     L4642  ; 進料分流右側昇降上定點
      AND     L4660  ; 右IR輸送進框補助下降定點
      AND     L53  ; 允許進料分流右側昇降下降
      AND     B1180  ; 右進料IR輸送暫停
      OUT     T353 D105  ; 自動進料分流右昇降  下降延遲
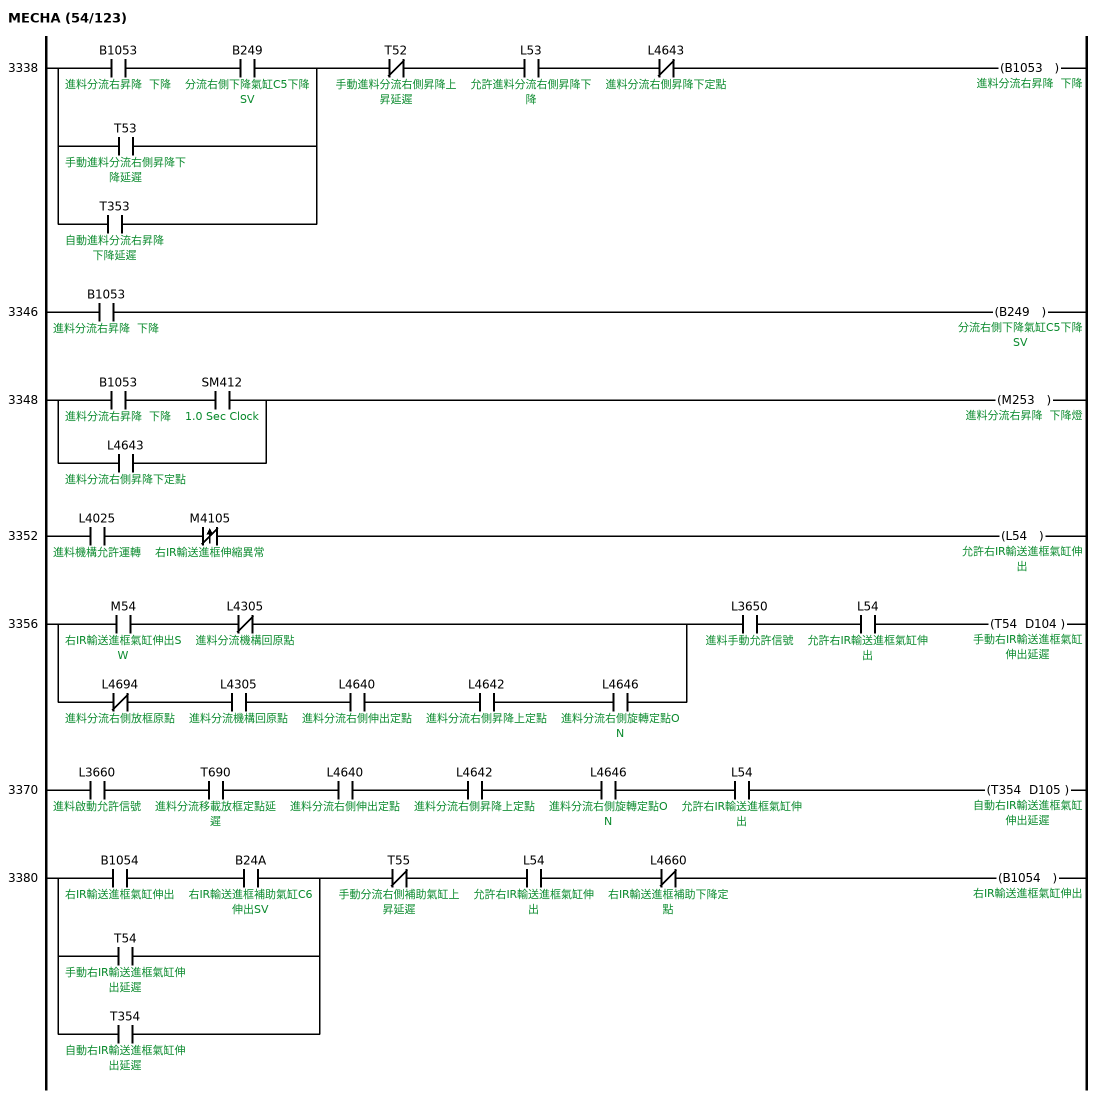
3338  LD      B1053  ; 進料分流右昇降  下降
      AND     B249  ; 分流右側下降氣缸C5下降SV
      OR      T53  ; 手動進料分流右側昇降下降延遲
      OR      T353  ; 自動進料分流右昇降  下降延遲
      ANI     T52  ; 手動進料分流右側昇降上昇延遲
      AND     L53  ; 允許進料分流右側昇降下降
      ANI     L4643  ; 進料分流右側昇降下定點
      OUT     B1053  ; 進料分流右昇降  下降
3346  LD      B1053  ; 進料分流右昇降  下降
      OUT     B249  ; 分流右側下降氣缸C5下降SV
3348  LD      B1053  ; 進料分流右昇降  下降
      AND     SM412  ; 1.0 Sec Clock
      OR      L4643  ; 進料分流右側昇降下定點
      OUT     M253  ; 進料分流右昇降  下降燈
3352  LD      L4025  ; 進料機構允許運轉
      ANDPI   M4105  ; 右IR輸送進框伸縮異常
      OUT     L54  ; 允許右IR輸送進框氣缸伸出
3356  LD      M54  ; 右IR輸送進框氣缸伸出SW
      ANI     L4305  ; 進料分流機構回原點
      LDI     L4694  ; 進料分流右側放框原點
      AND     L4305  ; 進料分流機構回原點
      AND     L4640  ; 進料分流右側伸出定點
      AND     L4642  ; 進料分流右側昇降上定點
      AND     L4646  ; 進料分流右側旋轉定點ON
      ORB
      AND     L3650  ; 進料手動允許信號
      AND     L54  ; 允許右IR輸送進框氣缸伸出
      OUT     T54 D104  ; 手動右IR輸送進框氣缸伸出延遲
3370  LD      L3660  ; 進料啟動允許信號
      AND     T690  ; 進料分流移載放框定點延遲
      AND     L4640  ; 進料分流右側伸出定點
      AND     L4642  ; 進料分流右側昇降上定點
      AND     L4646  ; 進料分流右側旋轉定點ON
      AND     L54  ; 允許右IR輸送進框氣缸伸出
      OUT     T354 D105  ; 自動右IR輸送進框氣缸伸出延遲
3380  LD      B1054  ; 右IR輸送進框氣缸伸出
      AND     B24A  ; 右IR輸送進框補助氣缸C6伸出SV
      OR      T54  ; 手動右IR輸送進框氣缸伸出延遲
      OR      T354  ; 自動右IR輸送進框氣缸伸出延遲
      ANI     T55  ; 手動分流右側補助氣缸上昇延遲
      AND     L54  ; 允許右IR輸送進框氣缸伸出
      ANI     L4660  ; 右IR輸送進框補助下降定點
      OUT     B1054  ; 右IR輸送進框氣缸伸出
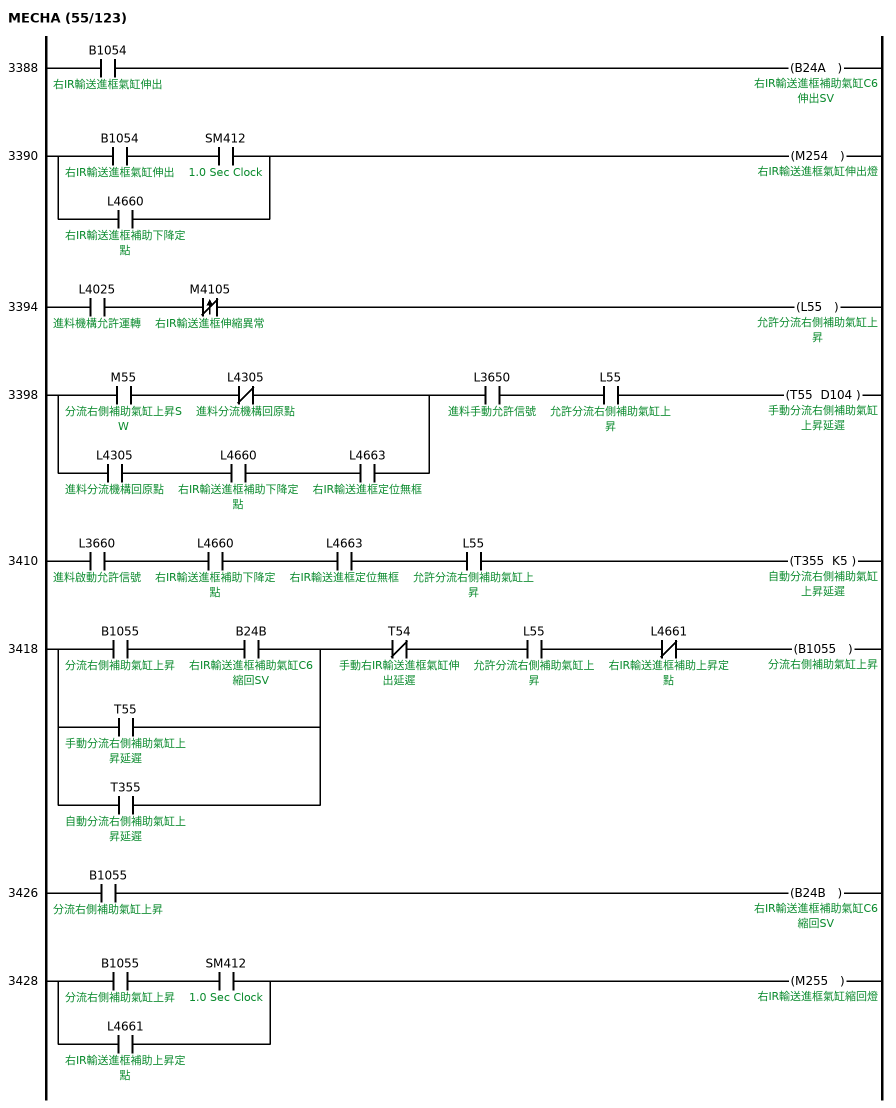
3388  LD      B1054  ; 右IR輸送進框氣缸伸出
      OUT     B24A  ; 右IR輸送進框補助氣缸C6伸出SV
3390  LD      B1054  ; 右IR輸送進框氣缸伸出
      AND     SM412  ; 1.0 Sec Clock
      OR      L4660  ; 右IR輸送進框補助下降定點
      OUT     M254  ; 右IR輸送進框氣缸伸出燈
3394  LD      L4025  ; 進料機構允許運轉
      ANDPI   M4105  ; 右IR輸送進框伸縮異常
      OUT     L55  ; 允許分流右側補助氣缸上昇
3398  LD      M55  ; 分流右側補助氣缸上昇SW
      ANI     L4305  ; 進料分流機構回原點
      LD      L4305  ; 進料分流機構回原點
      AND     L4660  ; 右IR輸送進框補助下降定點
      AND     L4663  ; 右IR輸送進框定位無框
      ORB
      AND     L3650  ; 進料手動允許信號
      AND     L55  ; 允許分流右側補助氣缸上昇
      OUT     T55 D104  ; 手動分流右側補助氣缸上昇延遲
3410  LD      L3660  ; 進料啟動允許信號
      AND     L4660  ; 右IR輸送進框補助下降定點
      AND     L4663  ; 右IR輸送進框定位無框
      AND     L55  ; 允許分流右側補助氣缸上昇
      OUT     T355 K5  ; 自動分流右側補助氣缸上昇延遲
3418  LD      B1055  ; 分流右側補助氣缸上昇
      AND     B24B  ; 右IR輸送進框補助氣缸C6縮回SV
      OR      T55  ; 手動分流右側補助氣缸上昇延遲
      OR      T355  ; 自動分流右側補助氣缸上昇延遲
      ANI     T54  ; 手動右IR輸送進框氣缸伸出延遲
      AND     L55  ; 允許分流右側補助氣缸上昇
      ANI     L4661  ; 右IR輸送進框補助上昇定點
      OUT     B1055  ; 分流右側補助氣缸上昇
3426  LD      B1055  ; 分流右側補助氣缸上昇
      OUT     B24B  ; 右IR輸送進框補助氣缸C6縮回SV
3428  LD      B1055  ; 分流右側補助氣缸上昇
      AND     SM412  ; 1.0 Sec Clock
      OR      L4661  ; 右IR輸送進框補助上昇定點
      OUT     M255  ; 右IR輸送進框氣缸縮回燈
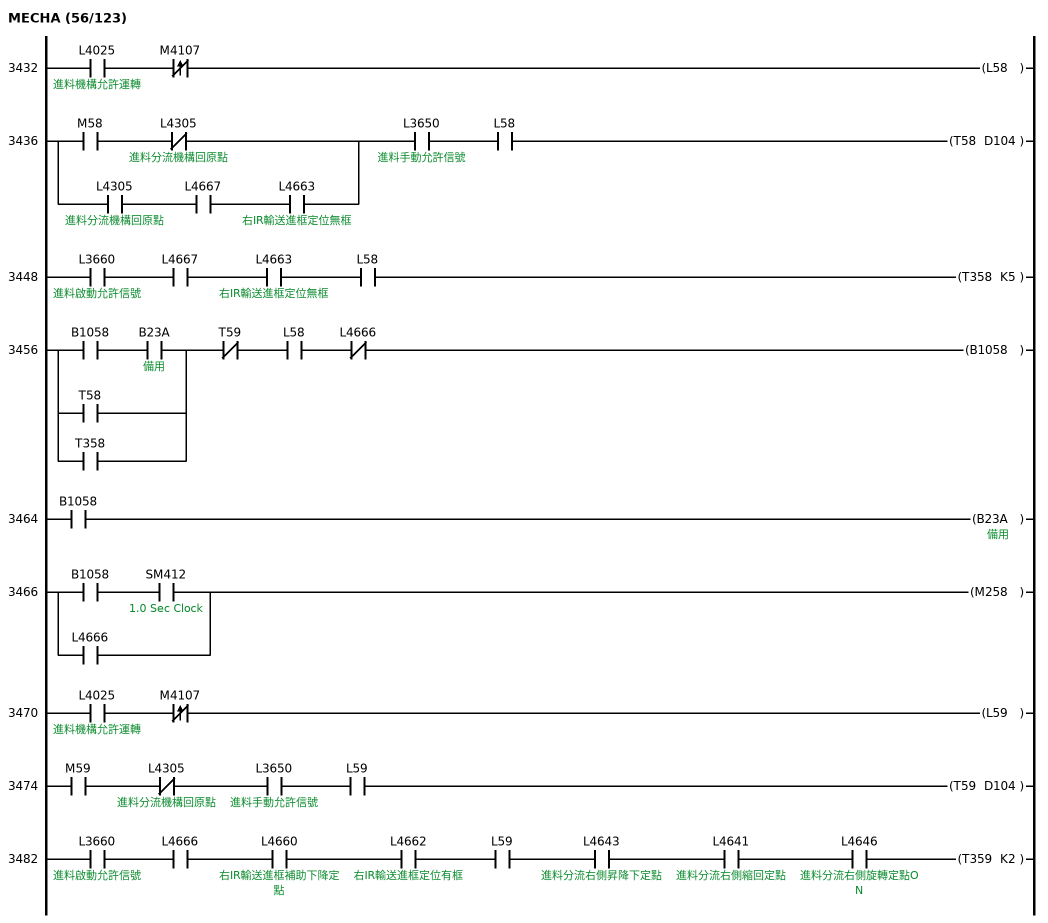
3432  LD      L4025  ; 進料機構允許運轉
      ANDPI   M4107
      OUT     L58
3436  LD      M58
      ANI     L4305  ; 進料分流機構回原點
      LD      L4305  ; 進料分流機構回原點
      AND     L4667
      AND     L4663  ; 右IR輸送進框定位無框
      ORB
      AND     L3650  ; 進料手動允許信號
      AND     L58
      OUT     T58 D104
3448  LD      L3660  ; 進料啟動允許信號
      AND     L4667
      AND     L4663  ; 右IR輸送進框定位無框
      AND     L58
      OUT     T358 K5
3456  LD      B1058
      AND     B23A  ; 備用
      OR      T58
      OR      T358
      ANI     T59
      AND     L58
      ANI     L4666
      OUT     B1058
3464  LD      B1058
      OUT     B23A  ; 備用
3466  LD      B1058
      AND     SM412  ; 1.0 Sec Clock
      OR      L4666
      OUT     M258
3470  LD      L4025  ; 進料機構允許運轉
      ANDPI   M4107
      OUT     L59
3474  LD      M59
      ANI     L4305  ; 進料分流機構回原點
      AND     L3650  ; 進料手動允許信號
      AND     L59
      OUT     T59 D104
3482  LD      L3660  ; 進料啟動允許信號
      AND     L4666
      AND     L4660  ; 右IR輸送進框補助下降定點
      AND     L4662  ; 右IR輸送進框定位有框
      AND     L59
      AND     L4643  ; 進料分流右側昇降下定點
      AND     L4641  ; 進料分流右側縮回定點
      AND     L4646  ; 進料分流右側旋轉定點ON
      OUT     T359 K2
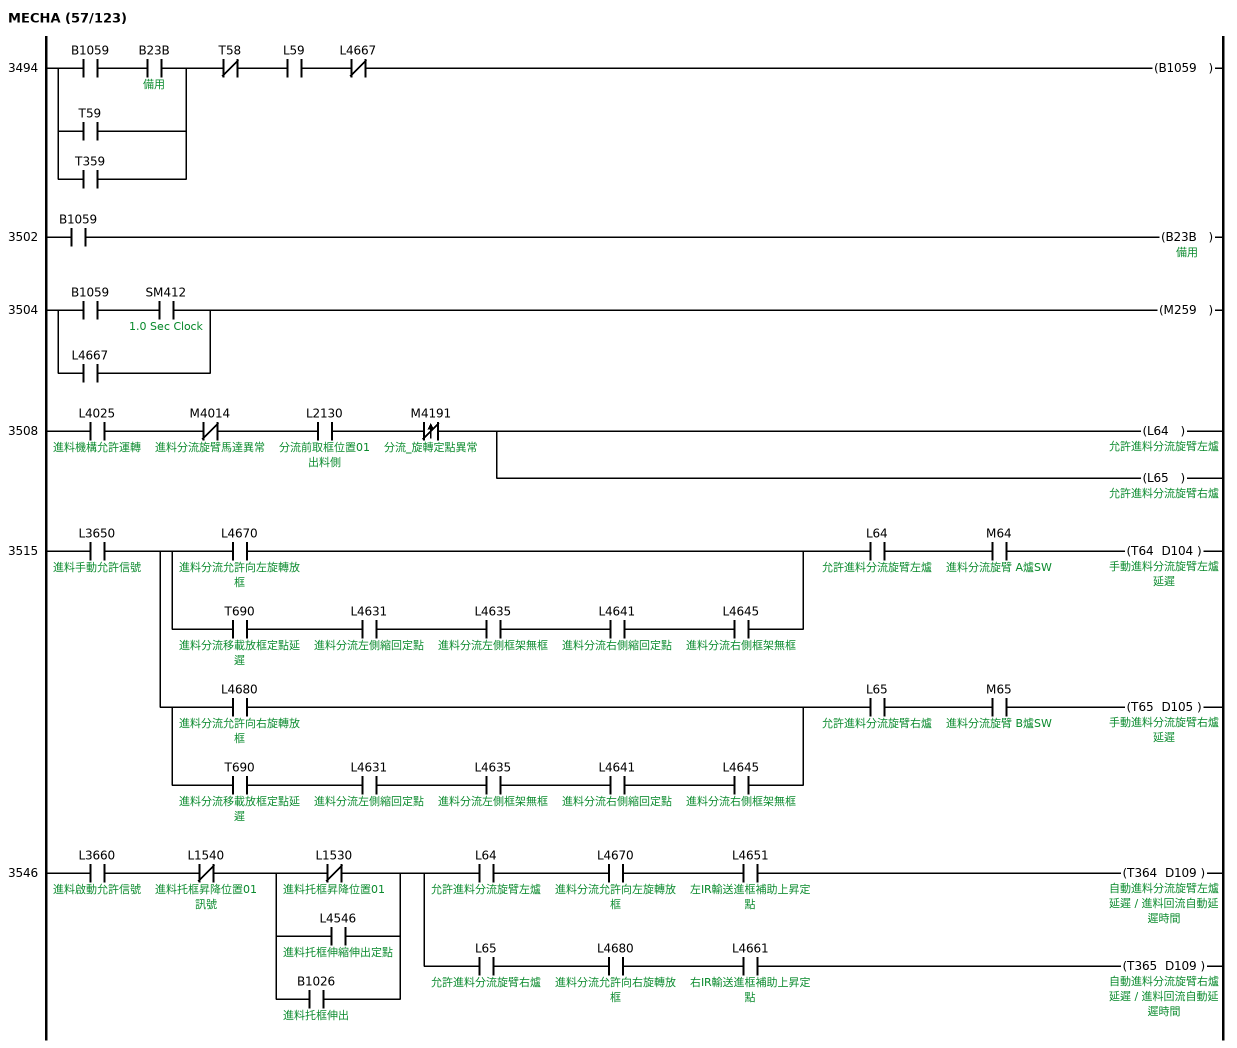
3494  LD      B1059
      AND     B23B  ; 備用
      OR      T59
      OR      T359
      ANI     T58
      AND     L59
      ANI     L4667
      OUT     B1059
3502  LD      B1059
      OUT     B23B  ; 備用
3504  LD      B1059
      AND     SM412  ; 1.0 Sec Clock
      OR      L4667
      OUT     M259
3508  LD      L4025  ; 進料機構允許運轉
      ANI     M4014  ; 進料分流旋臂馬達異常
      AND     L2130  ; 分流前取框位置01  出料側
      ANDPI   M4191  ; 分流_旋轉定點異常
      OUT     L64  ; 允許進料分流旋臂左爐
      OUT     L65  ; 允許進料分流旋臂右爐
3515  LD      L3650  ; 進料手動允許信號
      MPS
      LD      L4670  ; 進料分流允許向左旋轉放框
      LD      T690  ; 進料分流移載放框定點延遲
      AND     L4631  ; 進料分流左側縮回定點
      AND     L4635  ; 進料分流左側框架無框
      AND     L4641  ; 進料分流右側縮回定點
      AND     L4645  ; 進料分流右側框架無框
      ORB
      ANB
      AND     L64  ; 允許進料分流旋臂左爐
      AND     M64  ; 進料分流旋臂 A爐SW
      OUT     T64 D104  ; 手動進料分流旋臂左爐延遲
      MPP
      LD      L4680  ; 進料分流允許向右旋轉放框
      LD      T690  ; 進料分流移載放框定點延遲
      AND     L4631  ; 進料分流左側縮回定點
      AND     L4635  ; 進料分流左側框架無框
      AND     L4641  ; 進料分流右側縮回定點
      AND     L4645  ; 進料分流右側框架無框
      ORB
      ANB
      AND     L65  ; 允許進料分流旋臂右爐
      AND     M65  ; 進料分流旋臂 B爐SW
      OUT     T65 D105  ; 手動進料分流旋臂右爐延遲
3546  LD      L3660  ; 進料啟動允許信號
      ANI     L1540  ; 進料托框昇降位置01 訊號
      LDI     L1530  ; 進料托框昇降位置01
      OR      L4546  ; 進料托框伸縮伸出定點
      OR      B1026  ; 進料托框伸出
      ANB
      MPS
      AND     L64  ; 允許進料分流旋臂左爐
      AND     L4670  ; 進料分流允許向左旋轉放框
      AND     L4651  ; 左IR輸送進框補助上昇定點
      OUT     T364 D109  ; 自動進料分流旋臂左爐延遲 / 進料回流自動延遲時間
      MPP
      AND     L65  ; 允許進料分流旋臂右爐
      AND     L4680  ; 進料分流允許向右旋轉放框
      AND     L4661  ; 右IR輸送進框補助上昇定點
      OUT     T365 D109  ; 自動進料分流旋臂右爐延遲 / 進料回流自動延遲時間
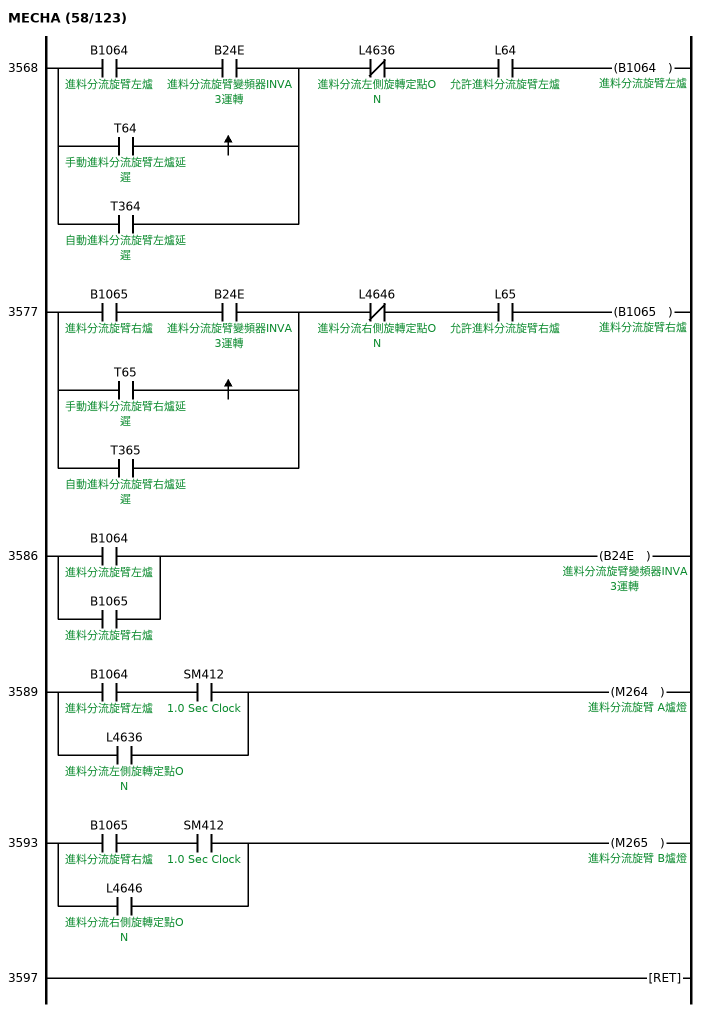
3568  LD      B1064  ; 進料分流旋臂左爐
      AND     B24E  ; 進料分流旋臂變頻器INVA3運轉
      LD      T64  ; 手動進料分流旋臂左爐延遲
      MEP
      ORB
      OR      T364  ; 自動進料分流旋臂左爐延遲
      ANI     L4636  ; 進料分流左側旋轉定點ON
      AND     L64  ; 允許進料分流旋臂左爐
      OUT     B1064  ; 進料分流旋臂左爐
3577  LD      B1065  ; 進料分流旋臂右爐
      AND     B24E  ; 進料分流旋臂變頻器INVA3運轉
      LD      T65  ; 手動進料分流旋臂右爐延遲
      MEP
      ORB
      OR      T365  ; 自動進料分流旋臂右爐延遲
      ANI     L4646  ; 進料分流右側旋轉定點ON
      AND     L65  ; 允許進料分流旋臂右爐
      OUT     B1065  ; 進料分流旋臂右爐
3586  LD      B1064  ; 進料分流旋臂左爐
      OR      B1065  ; 進料分流旋臂右爐
      OUT     B24E  ; 進料分流旋臂變頻器INVA3運轉
3589  LD      B1064  ; 進料分流旋臂左爐
      AND     SM412  ; 1.0 Sec Clock
      OR      L4636  ; 進料分流左側旋轉定點ON
      OUT     M264  ; 進料分流旋臂 A爐燈
3593  LD      B1065  ; 進料分流旋臂右爐
      AND     SM412  ; 1.0 Sec Clock
      OR      L4646  ; 進料分流右側旋轉定點ON
      OUT     M265  ; 進料分流旋臂 B爐燈
3597  RET
      P1031
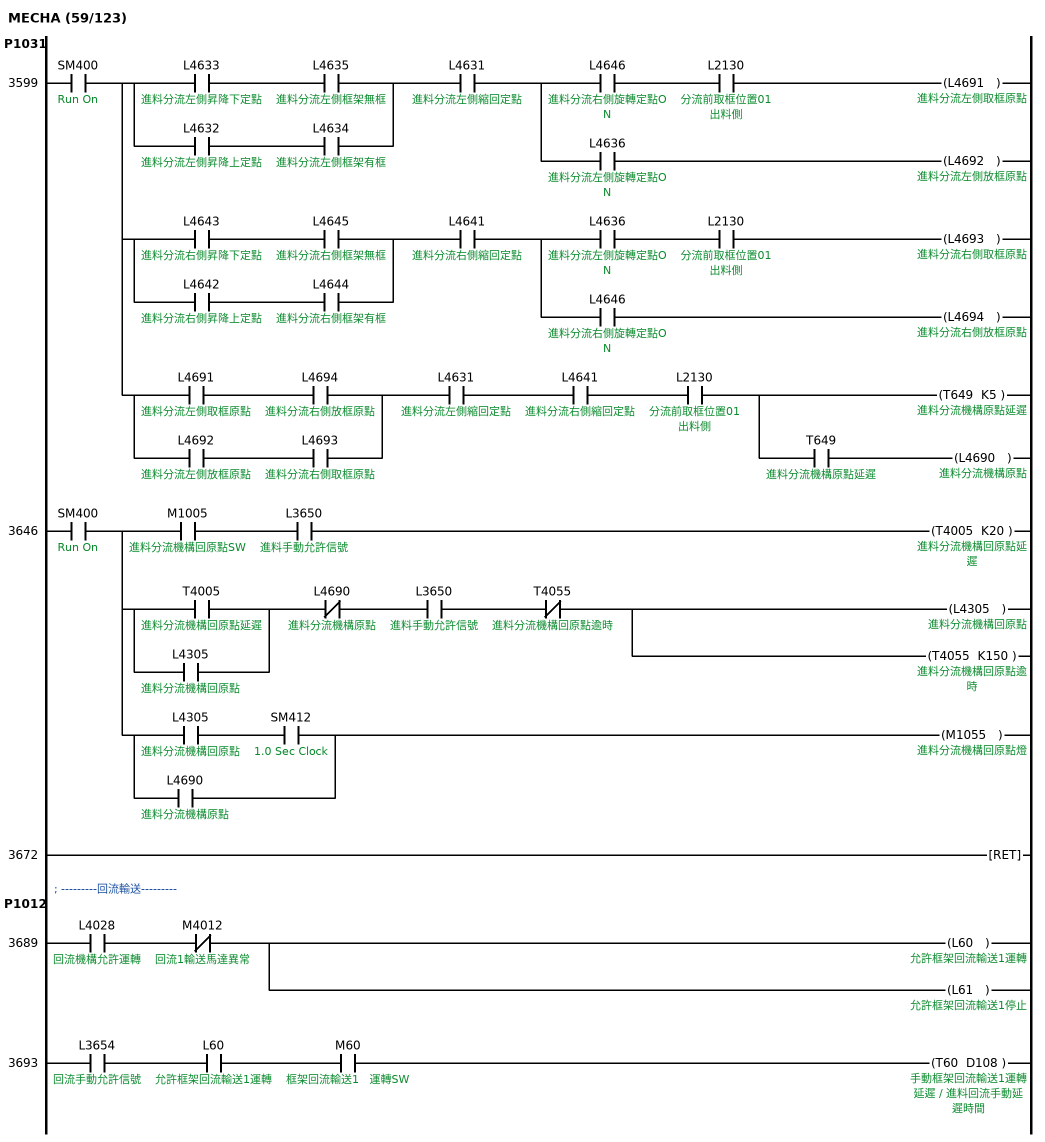
3599  LD      SM400  ; Run On
      MPS
      LD      L4633  ; 進料分流左側昇降下定點
      AND     L4635  ; 進料分流左側框架無框
      LD      L4632  ; 進料分流左側昇降上定點
      AND     L4634  ; 進料分流左側框架有框
      ORB
      ANB
      AND     L4631  ; 進料分流左側縮回定點
      MPS
      AND     L4646  ; 進料分流右側旋轉定點ON
      AND     L2130  ; 分流前取框位置01  出料側
      OUT     L4691  ; 進料分流左側取框原點
      MPP
      AND     L4636  ; 進料分流左側旋轉定點ON
      OUT     L4692  ; 進料分流左側放框原點
      MRD
      LD      L4643  ; 進料分流右側昇降下定點
      AND     L4645  ; 進料分流右側框架無框
      LD      L4642  ; 進料分流右側昇降上定點
      AND     L4644  ; 進料分流右側框架有框
      ORB
      ANB
      AND     L4641  ; 進料分流右側縮回定點
      MPS
      AND     L4636  ; 進料分流左側旋轉定點ON
      AND     L2130  ; 分流前取框位置01  出料側
      OUT     L4693  ; 進料分流右側取框原點
      MPP
      AND     L4646  ; 進料分流右側旋轉定點ON
      OUT     L4694  ; 進料分流右側放框原點
      MPP
      LD      L4691  ; 進料分流左側取框原點
      AND     L4694  ; 進料分流右側放框原點
      LD      L4692  ; 進料分流左側放框原點
      AND     L4693  ; 進料分流右側取框原點
      ORB
      ANB
      AND     L4631  ; 進料分流左側縮回定點
      AND     L4641  ; 進料分流右側縮回定點
      AND     L2130  ; 分流前取框位置01  出料側
      OUT     T649 K5  ; 進料分流機構原點延遲
      AND     T649  ; 進料分流機構原點延遲
      OUT     L4690  ; 進料分流機構原點
3646  LD      SM400  ; Run On
      MPS
      AND     M1005  ; 進料分流機構回原點SW
      AND     L3650  ; 進料手動允許信號
      OUT     T4005 K20  ; 進料分流機構回原點延遲
      MRD
      LD      T4005  ; 進料分流機構回原點延遲
      OR      L4305  ; 進料分流機構回原點
      ANB
      ANI     L4690  ; 進料分流機構原點
      AND     L3650  ; 進料手動允許信號
      ANI     T4055  ; 進料分流機構回原點逾時
      OUT     L4305  ; 進料分流機構回原點
      OUT     T4055 K150  ; 進料分流機構回原點逾時
      MPP
      LD      L4305  ; 進料分流機構回原點
      AND     SM412  ; 1.0 Sec Clock
      OR      L4690  ; 進料分流機構原點
      ANB
      OUT     M1055  ; 進料分流機構回原點燈
3672  RET
; ---------回流輸送---------
      P1012
3689  LD      L4028  ; 回流機構允許運轉
      ANI     M4012  ; 回流1輸送馬達異常
      OUT     L60  ; 允許框架回流輸送1運轉
      OUT     L61  ; 允許框架回流輸送1停止
3693  LD      L3654  ; 回流手動允許信號
      AND     L60  ; 允許框架回流輸送1運轉
      AND     M60  ; 框架回流輸送1   運轉SW
      OUT     T60 D108  ; 手動框架回流輸送1運轉延遲 / 進料回流手動延遲時間
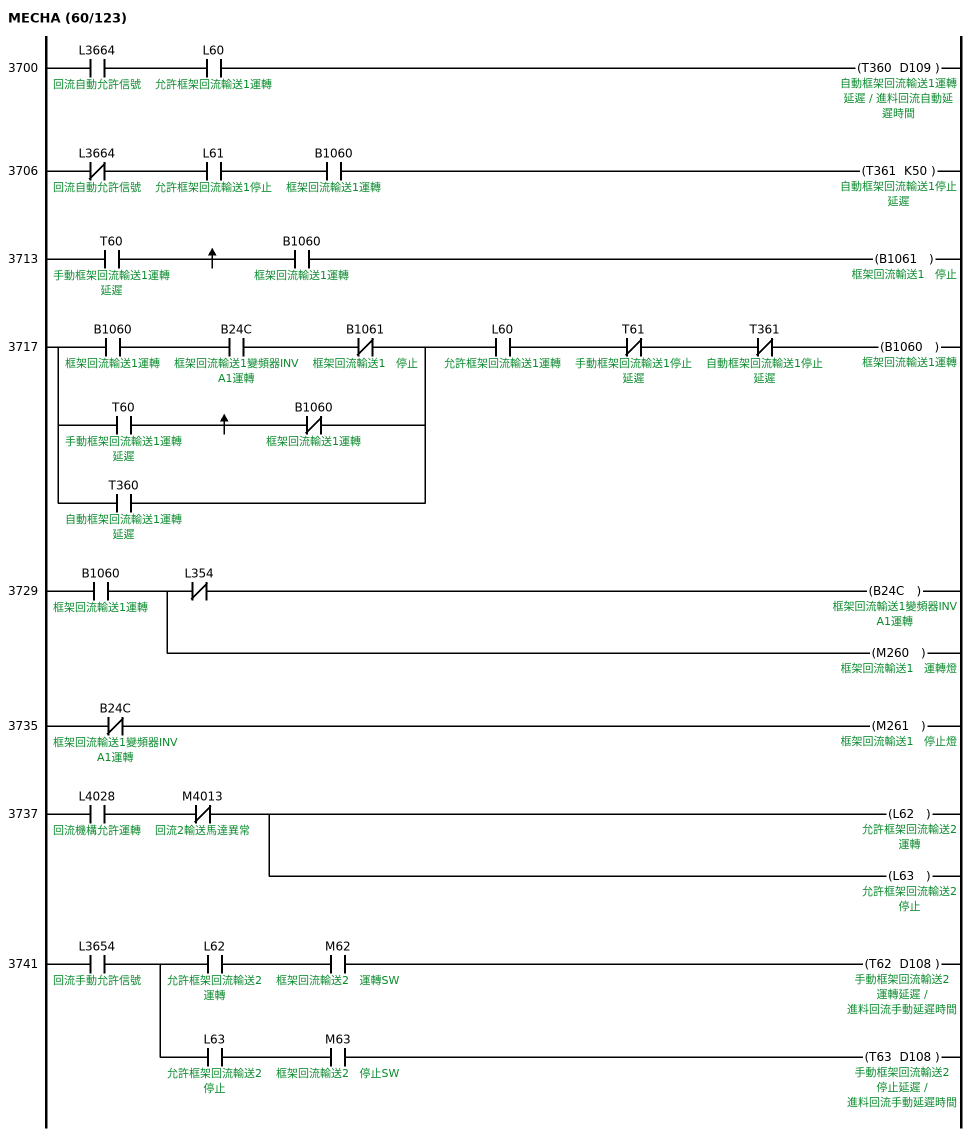
3700  LD      L3664  ; 回流自動允許信號
      AND     L60  ; 允許框架回流輸送1運轉
      OUT     T360 D109  ; 自動框架回流輸送1運轉延遲 / 進料回流自動延遲時間
3706  LDI     L3664  ; 回流自動允許信號
      AND     L61  ; 允許框架回流輸送1停止
      AND     B1060  ; 框架回流輸送1運轉
      OUT     T361 K50  ; 自動框架回流輸送1停止延遲
3713  LD      T60  ; 手動框架回流輸送1運轉延遲
      MEP
      AND     B1060  ; 框架回流輸送1運轉
      OUT     B1061  ; 框架回流輸送1   停止
3717  LD      B1060  ; 框架回流輸送1運轉
      AND     B24C  ; 框架回流輸送1變頻器INVA1運轉
      ANI     B1061  ; 框架回流輸送1   停止
      LD      T60  ; 手動框架回流輸送1運轉延遲
      MEP
      ANI     B1060  ; 框架回流輸送1運轉
      ORB
      OR      T360  ; 自動框架回流輸送1運轉延遲
      AND     L60  ; 允許框架回流輸送1運轉
      ANI     T61  ; 手動框架回流輸送1停止延遲
      ANI     T361  ; 自動框架回流輸送1停止延遲
      OUT     B1060  ; 框架回流輸送1運轉
3729  LD      B1060  ; 框架回流輸送1運轉
      MPS
      ANI     L354
      OUT     B24C  ; 框架回流輸送1變頻器INVA1運轉
      MPP
      OUT     M260  ; 框架回流輸送1   運轉燈
3735  LDI     B24C  ; 框架回流輸送1變頻器INVA1運轉
      OUT     M261  ; 框架回流輸送1   停止燈
3737  LD      L4028  ; 回流機構允許運轉
      ANI     M4013  ; 回流2輸送馬達異常
      OUT     L62  ; 允許框架回流輸送2   運轉
      OUT     L63  ; 允許框架回流輸送2   停止
3741  LD      L3654  ; 回流手動允許信號
      MPS
      AND     L62  ; 允許框架回流輸送2   運轉
      AND     M62  ; 框架回流輸送2   運轉SW
      OUT     T62 D108  ; 手動框架回流輸送2   運轉延遲 / 進料回流手動延遲時間
      MPP
      AND     L63  ; 允許框架回流輸送2   停止
      AND     M63  ; 框架回流輸送2   停止SW
      OUT     T63 D108  ; 手動框架回流輸送2   停止延遲 / 進料回流手動延遲時間
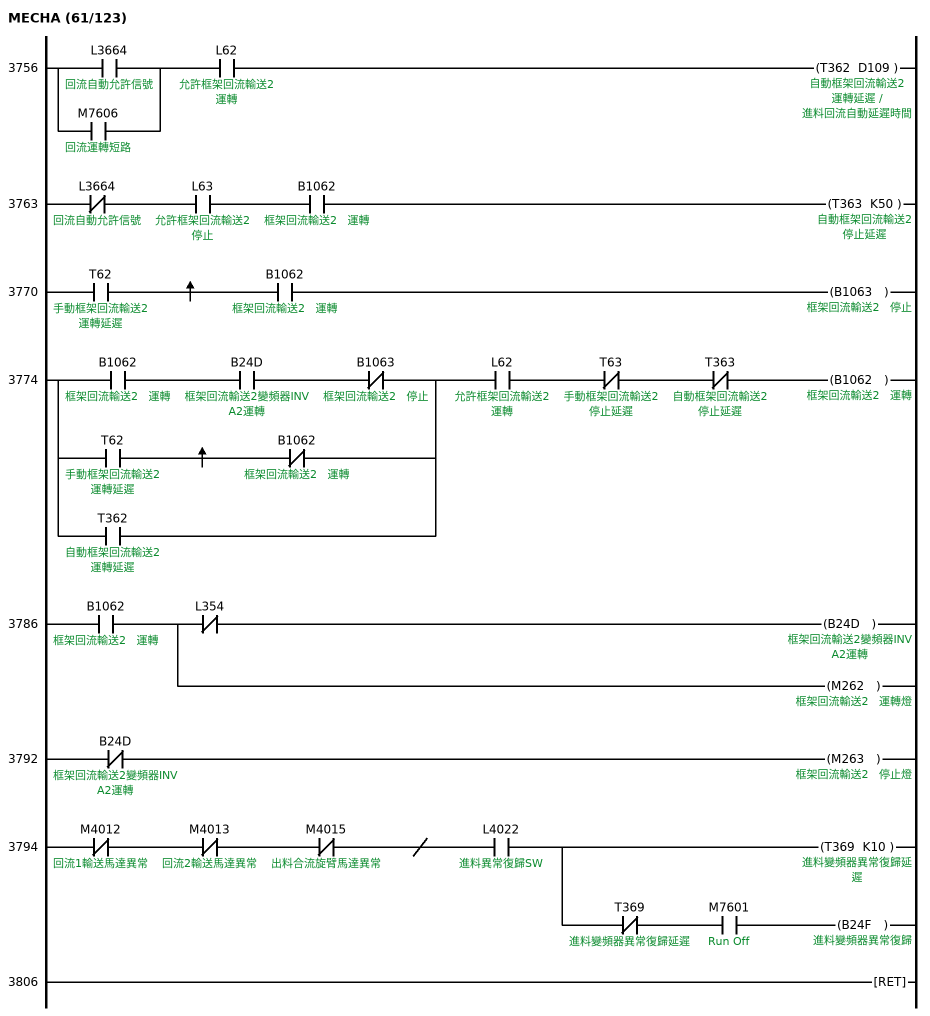
3756  LD      L3664  ; 回流自動允許信號
      OR      M7606  ; 回流運轉短路
      AND     L62  ; 允許框架回流輸送2   運轉
      OUT     T362 D109  ; 自動框架回流輸送2   運轉延遲 / 進料回流自動延遲時間
3763  LDI     L3664  ; 回流自動允許信號
      AND     L63  ; 允許框架回流輸送2   停止
      AND     B1062  ; 框架回流輸送2   運轉
      OUT     T363 K50  ; 自動框架回流輸送2   停止延遲
3770  LD      T62  ; 手動框架回流輸送2   運轉延遲
      MEP
      AND     B1062  ; 框架回流輸送2   運轉
      OUT     B1063  ; 框架回流輸送2   停止
3774  LD      B1062  ; 框架回流輸送2   運轉
      AND     B24D  ; 框架回流輸送2變頻器INVA2運轉
      ANI     B1063  ; 框架回流輸送2   停止
      LD      T62  ; 手動框架回流輸送2   運轉延遲
      MEP
      ANI     B1062  ; 框架回流輸送2   運轉
      ORB
      OR      T362  ; 自動框架回流輸送2   運轉延遲
      AND     L62  ; 允許框架回流輸送2   運轉
      ANI     T63  ; 手動框架回流輸送2   停止延遲
      ANI     T363  ; 自動框架回流輸送2   停止延遲
      OUT     B1062  ; 框架回流輸送2   運轉
3786  LD      B1062  ; 框架回流輸送2   運轉
      MPS
      ANI     L354
      OUT     B24D  ; 框架回流輸送2變頻器INVA2運轉
      MPP
      OUT     M262  ; 框架回流輸送2   運轉燈
3792  LDI     B24D  ; 框架回流輸送2變頻器INVA2運轉
      OUT     M263  ; 框架回流輸送2   停止燈
3794  LDI     M4012  ; 回流1輸送馬達異常
      ANI     M4013  ; 回流2輸送馬達異常
      ANI     M4015  ; 出料合流旋臂馬達異常
      INV
      AND     L4022  ; 進料異常復歸SW
      OUT     T369 K10  ; 進料變頻器異常復歸延遲
      ANI     T369  ; 進料變頻器異常復歸延遲
      AND     M7601  ; Run Off
      OUT     B24F  ; 進料變頻器異常復歸
3806  RET
; --------出料機構-----------
      P1040
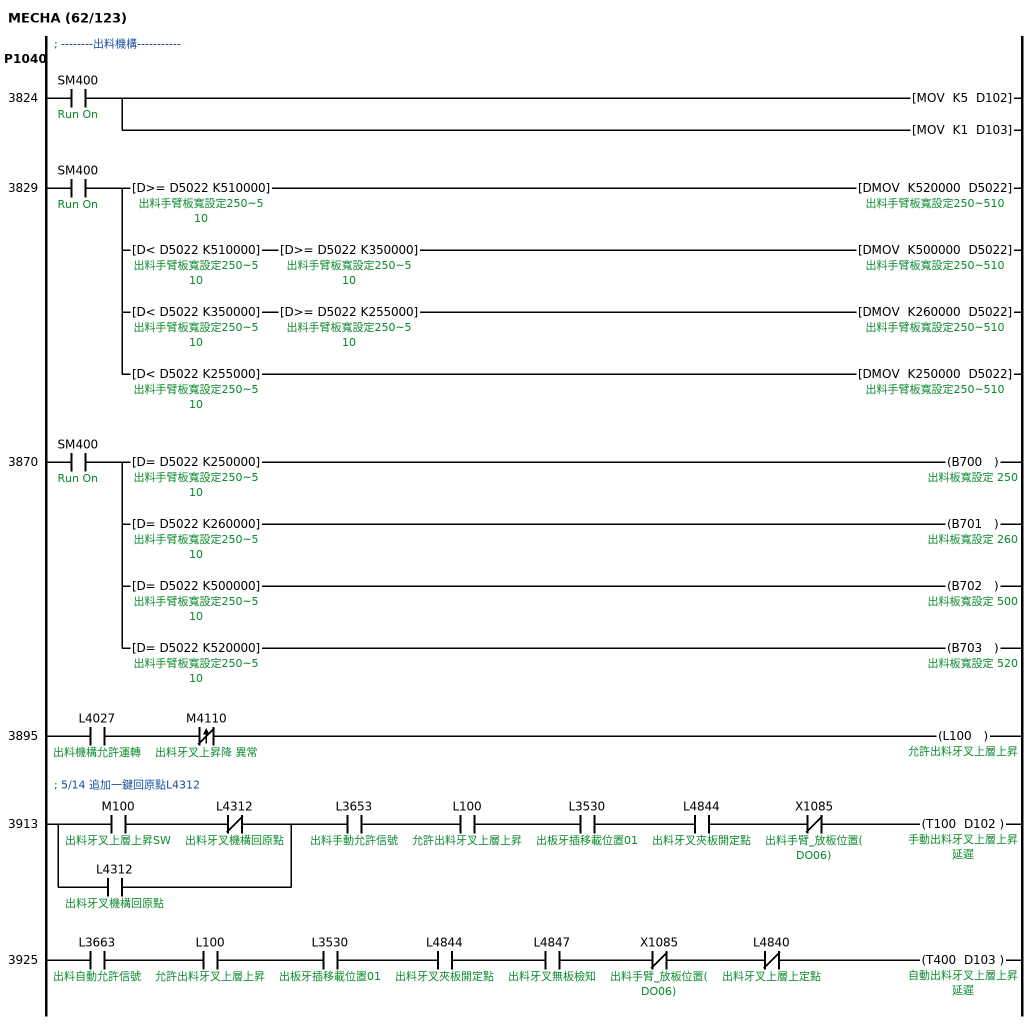
3824  LD      SM400  ; Run On
      MOV     K5 D102
      MOV     K1 D103
3829  LD      SM400  ; Run On
      MPS
      ANDD>=  D5022 K510000  ; 出料手臂板寬設定250~510
      DMOV    K520000 D5022
      MRD
      ANDD<   D5022 K510000  ; 出料手臂板寬設定250~510
      ANDD>=  D5022 K350000  ; 出料手臂板寬設定250~510
      DMOV    K500000 D5022
      MRD
      ANDD<   D5022 K350000  ; 出料手臂板寬設定250~510
      ANDD>=  D5022 K255000  ; 出料手臂板寬設定250~510
      DMOV    K260000 D5022
      MPP
      ANDD<   D5022 K255000  ; 出料手臂板寬設定250~510
      DMOV    K250000 D5022
3870  LD      SM400  ; Run On
      MPS
      ANDD=   D5022 K250000  ; 出料手臂板寬設定250~510
      OUT     B700  ; 出料板寬設定 250
      MRD
      ANDD=   D5022 K260000  ; 出料手臂板寬設定250~510
      OUT     B701  ; 出料板寬設定 260
      MRD
      ANDD=   D5022 K500000  ; 出料手臂板寬設定250~510
      OUT     B702  ; 出料板寬設定 500
      MPP
      ANDD=   D5022 K520000  ; 出料手臂板寬設定250~510
      OUT     B703  ; 出料板寬設定 520
3895  LD      L4027  ; 出料機構允許運轉
      ANDPI   M4110  ; 出料牙叉上昇降 異常
      OUT     L100  ; 允許出料牙叉上層上昇
; 5/14 追加一鍵回原點L4312
3913  LD      M100  ; 出料牙叉上層上昇SW
      ANI     L4312  ; 出料牙叉機構回原點
      OR      L4312  ; 出料牙叉機構回原點
      AND     L3653  ; 出料手動允許信號
      AND     L100  ; 允許出料牙叉上層上昇
      AND     L3530  ; 出板牙插移載位置01
      AND     L4844  ; 出料牙叉夾板開定點
      ANI     X1085  ; 出料手臂_放板位置(DO06)
      OUT     T100 D102  ; 手動出料牙叉上層上昇延遲
3925  LD      L3663  ; 出料自動允許信號
      AND     L100  ; 允許出料牙叉上層上昇
      AND     L3530  ; 出板牙插移載位置01
      AND     L4844  ; 出料牙叉夾板開定點
      AND     L4847  ; 出料牙叉無板檢知
      ANI     X1085  ; 出料手臂_放板位置(DO06)
      ANI     L4840  ; 出料牙叉上層上定點
      OUT     T400 D103  ; 自動出料牙叉上層上昇延遲
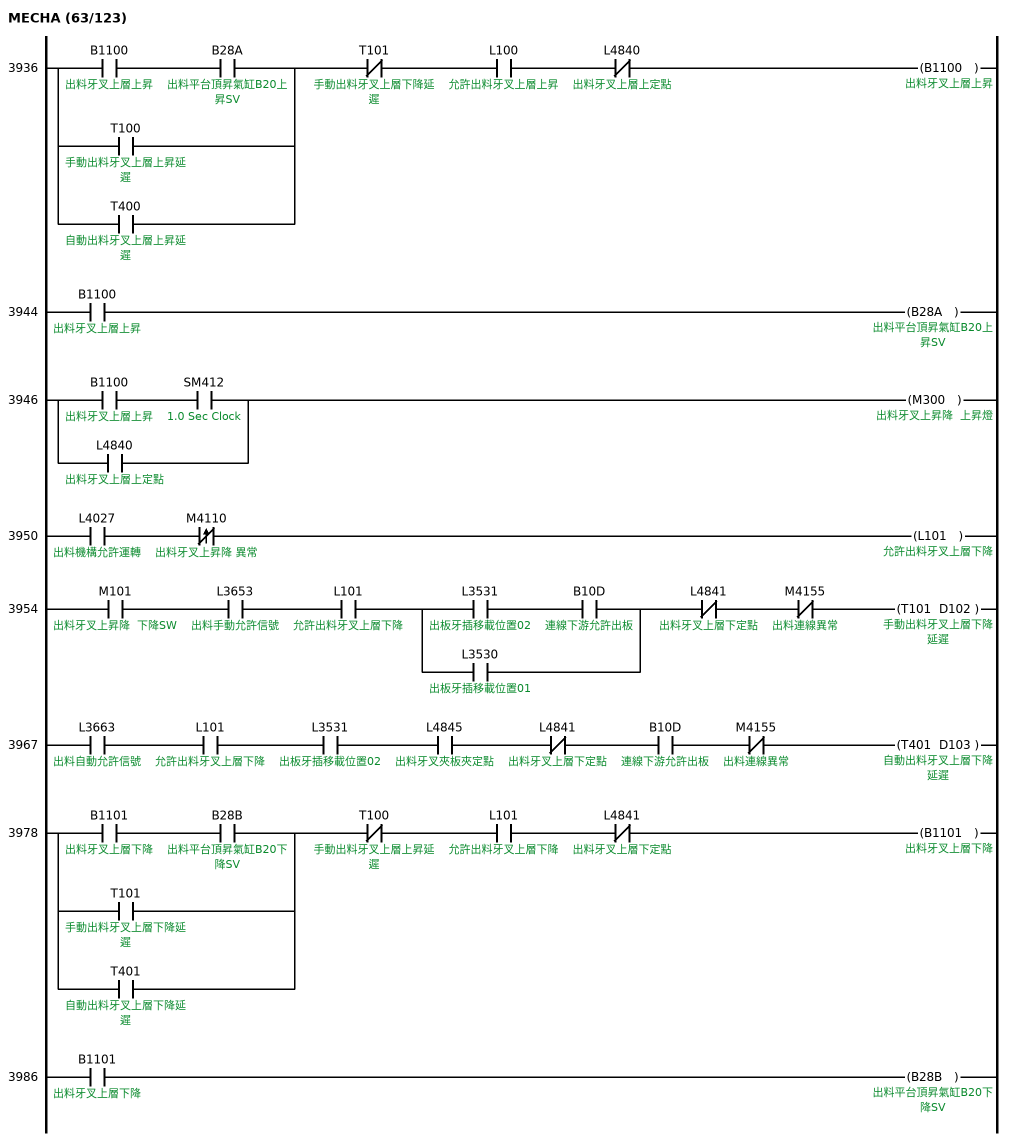
3936  LD      B1100  ; 出料牙叉上層上昇
      AND     B28A  ; 出料平台頂昇氣缸B20上昇SV
      OR      T100  ; 手動出料牙叉上層上昇延遲
      OR      T400  ; 自動出料牙叉上層上昇延遲
      ANI     T101  ; 手動出料牙叉上層下降延遲
      AND     L100  ; 允許出料牙叉上層上昇
      ANI     L4840  ; 出料牙叉上層上定點
      OUT     B1100  ; 出料牙叉上層上昇
3944  LD      B1100  ; 出料牙叉上層上昇
      OUT     B28A  ; 出料平台頂昇氣缸B20上昇SV
3946  LD      B1100  ; 出料牙叉上層上昇
      AND     SM412  ; 1.0 Sec Clock
      OR      L4840  ; 出料牙叉上層上定點
      OUT     M300  ; 出料牙叉上昇降  上昇燈
3950  LD      L4027  ; 出料機構允許運轉
      ANDPI   M4110  ; 出料牙叉上昇降 異常
      OUT     L101  ; 允許出料牙叉上層下降
3954  LD      M101  ; 出料牙叉上昇降  下降SW
      AND     L3653  ; 出料手動允許信號
      AND     L101  ; 允許出料牙叉上層下降
      LD      L3531  ; 出板牙插移載位置02
      AND     B10D  ; 連線下游允許出板
      OR      L3530  ; 出板牙插移載位置01
      ANB
      ANI     L4841  ; 出料牙叉上層下定點
      ANI     M4155  ; 出料連線異常
      OUT     T101 D102  ; 手動出料牙叉上層下降延遲
3967  LD      L3663  ; 出料自動允許信號
      AND     L101  ; 允許出料牙叉上層下降
      AND     L3531  ; 出板牙插移載位置02
      AND     L4845  ; 出料牙叉夾板夾定點
      ANI     L4841  ; 出料牙叉上層下定點
      AND     B10D  ; 連線下游允許出板
      ANI     M4155  ; 出料連線異常
      OUT     T401 D103  ; 自動出料牙叉上層下降延遲
3978  LD      B1101  ; 出料牙叉上層下降
      AND     B28B  ; 出料平台頂昇氣缸B20下降SV
      OR      T101  ; 手動出料牙叉上層下降延遲
      OR      T401  ; 自動出料牙叉上層下降延遲
      ANI     T100  ; 手動出料牙叉上層上昇延遲
      AND     L101  ; 允許出料牙叉上層下降
      ANI     L4841  ; 出料牙叉上層下定點
      OUT     B1101  ; 出料牙叉上層下降
3986  LD      B1101  ; 出料牙叉上層下降
      OUT     B28B  ; 出料平台頂昇氣缸B20下降SV
